// TIA Portal V19 program export: 0 tag tables, 0 data types, 8 data blocks, 13 code blocks (in call order from the OBs), 23 instance data blocks

DATA_BLOCK "AI SCALING DB"   // DB5
{ S7_Optimized_Access := 'TRUE' }
// stored: MemoryReserve 100
   VAR RETAIN
      MIN : Struct
         "SYRUP VESSEL TEMP SENSOR" : Real := -50.0;
         "PREMIXING VESSEL TEMP SENSOR" : Real := -50.0;
         "SUGAR VESSEL TEMP SENSOR" : Real := -50.0;
         "STEAM LINE_1 TEMP SENSOR" : Real := -50.0;
         "STEAM LINE_2 TEMP SENSOR" : Real := -50.0;
         "PRESSURE TRANSMITTER 1" : Real := -1.0;
         "PRESSURE TRANSMITTER 2" : Real := -1.0;
         "VACCIM TRANSMITTER 1" : Real := -750.0;
         "VACCIM TRANSMITTER 2" : Real := -750.0;
         "VACCUM TRANSMITTER 3" : Real := -750.0;
         "SYRUP LOAD CELL" : Real := 0.0;
         "PREMIXING LOAD CELL" : Real := 0.0;
         "SUGAR LOAD CELL" : Real := 0.0;
         "ULTRASONIC LEVEL SENSOR-1" : Real := 0.0;
         "ULTRASONIC LEVEL SENSOR-2" : Real := 0.0;
         "ULTRASONIC LEVEL SENSOR-3" : Real := 0.0;
      END_STRUCT;
      MAX : Struct
         "SYRUP VESSEL TEMP SENSOR" : Real := 250.0;
         "PREMIXING VESSEL TEMP SENSOR" : Real := 250.0;
         "SUGAR VESSEL TEMP SENSOR" : Real := 250.0;
         "STEAM LINE_1 TEMP SENSOR" : Real := 250.0;
         "STEAM LINE_2 TEMP SENSOR" : Real := 250.0;
         "PRESSURE TRANSMITTER 1" : Real := 5.0;
         "PRESSURE TRANSMITTER 2" : Real := 5.0;
         "VACCIM TRANSMITTER 1" : Real := 0.0;
         "VACCIM TRANSMITTER 2" : Real := 0.0;
         "VACCUM TRANSMITTER 3" : Real := 0.0;
         "SYRUP LOAD CELL" : Real := 5000.0;
         "PREMIXING LOAD CELL" : Real := 1500.0;
         "SUGAR LOAD CELL" : Real := 3750.0;
         "ULTRASONIC LEVEL SENSOR-1" : Real := 10000.0;
         "ULTRASONIC LEVEL SENSOR-2" : Real := 10000.0;
         "ULTRASONIC LEVEL SENSOR-3" : Real := 10000.0;
      END_STRUCT;
   END_VAR
   VAR
      PV : Struct
         "SYRUP VESSEL TEMP SENSOR" : Real;
         "PREMIXING VESSEL TEMP SENSOR" : Real;
         "SUGAR VESSEL TEMP SENSOR" : Real;
         "STEAM LINE_1 TEMP SENSOR" : Real;
         "STEAM LINE_2 TEMP SENSOR" : Real;
         "PRESSURE TRANSMITTER 1" : Real;
         "PRESSURE TRANSMITTER 2" : Real;
         "VACCIM TRANSMITTER 1" : Real;
         "VACCIM TRANSMITTER 2" : Real;
         "VACCUM TRANSMITTER 3" : Real;
         "SYRUP LOAD CELL" : Real;
         "PREMIXING LOAD CELL" : Real;
         "SUGAR LOAD CELL" : Real;
         "ULTRASONIC LEVEL SENSOR-1" : Real;
         "ULTRASONIC LEVEL SENSOR-2" : Real;
         "ULTRASONIC LEVEL SENSOR-3" : Real;
      END_STRUCT;
   END_VAR
BEGIN
END_DATA_BLOCK

DATA_BLOCK "AO SCALING DB"   // DB6
{ S7_Optimized_Access := 'TRUE' }
// stored: MemoryReserve 100
   VAR
      SET : Struct
         "SYRUP MFG VESSEL SPEED" : Real;
         "PREMIXING VESSEL SPEED" : Real;
         "SUGAR VESSEL SPEED" : Real;
         SPARE : Real;
      END_STRUCT;
   END_VAR
   VAR RETAIN
      MIN : Struct
         "SYRUP MFG VESSEL SPEED" : Real;
         "PREMIXING VESSEL SPEED" : Real;
         "SUGAR VESSEL SPEED" : Real;
         SPARE : Real;
      END_STRUCT;
      MAX : Struct
         "SYRUP MFG VESSEL SPEED" : Real := 1450.0;
         "PREMIXING VESSEL SPEED" : Real := 1450.0;
         "SUGAR VESSEL SPEED" : Real := 1450.0;
         SPARE : Real;
      END_STRUCT;
   END_VAR
   VAR
      PV : Struct
         "SYRUP MFG VESSEL SPEED" : Real;
         "PREMIXING VESSEL SPEED" : Real;
         "SUGAR VESSEL SPEED" : Real;
         SPARE : Real;
      END_STRUCT;
   END_VAR
BEGIN
END_DATA_BLOCK

DATA_BLOCK "DO MAPING"   // DB2
{ S7_Optimized_Access := 'TRUE' }
// stored: MemoryReserve 100
   VAR
      "SYRUP MFG VESSEL BOTTOM STERROR RUN" : Bool;
      "PREMIXING VESSEL BOTTOM STERROR RUN" : Bool;
      "INLINE 1 HOMOGENIZER MOTOR1 RUN" : Bool;
      "INLINE 2 HOMOGENIZER MOTOR 2 RUN" : Bool;
      "FILTER PRESS MOTOR 1 RUN" : Bool;
      "FILTER PRESS MOTOR 2 RUN" : Bool;
      "VACCUM PUMP MOTOR-W 1 RUN" : Bool;
      "VACCUMP PUMP MOTOR-S2 RUN" : Bool;
      "VACCUMP PUMP MOTOR-W 3 RUN" : Bool;
      "VACCUMP PUMP MOTOR-S 4 RUN" : Bool;
      "SUGAR VESSEL BOTTOM STERROR RUN" : Bool;
      "BASKET FILTER MOTOR RUN" : Bool;
      "PBV-01 INGREDIENT INLET" : Bool;
      "PBV-02 CIP INLET (SPRAY BALL)" : Bool;
      "PBV-03 VENT FILTER ISOLATION" : Bool;
      "PBV-04 PW INLET" : Bool;
      "PBV-07 PREMIX TANK DRAIN VALVE" : Bool;
      "PAV-09 JACKET STEAM INLET" : Bool;
      "PAV-10 JACKET CONDENSATE DRAIN" : Bool;
      "PAV-11 JACKET BYPASS DRAIN VALVE" : Bool;
      "PAV-12 SEAL COOLING INLET" : Bool;
      "PAV-13 WATER COOLING INLET" : Bool;
      "PAV-14 WATER COOLING OUTLET" : Bool;
      "PBV-15 VACUUM INLET" : Bool;
      "PBV-16 VACUUM VENT VALVE" : Bool;
      "PFBV-17 TANK OUTLET VALVE" : Bool;
      "PBV-19 PW INLET" : Bool;
      "PBV-20 CIP INLET (SPRAY BALL)" : Bool;
      "PBV-21 VENT FILTER ISOLATION" : Bool;
      "PBV-22 INGREDIENT INLET (SUGAR INLET)" : Bool;
      "PBV-25 BOTTOM OUTLET TO DRAIN VALVE" : Bool;
      "PAV-27 JACKET STEAM INLET" : Bool;
      "PAV-28 SEAL COOLING INLET" : Bool;
      "PAV-29 JACKET CONDENSATE DRAIN" : Bool;
      "PBV-30 VACUUM INLET VALVE" : Bool;
      "PBV-31 VACUUM VENT VALVE" : Bool;
      "PFBV-32 TANK OUTLET VALVE" : Bool;
      "PBV-36 PW INLET" : Bool;
      "PBV-37 VENT FILTER ISOLATION" : Bool;
      "PBV-38 CIP INLET LINE" : Bool;
      "PBV-41 MFG TANK DRAIN VALVE" : Bool;
      "PAV-50 JACKET STEAM INLET" : Bool;
      "PAV-51 WATER COOLING OUTLET" : Bool;
      "PAV-52 WATER COOLING INLET" : Bool;
      "PAV-53 SEAL COOLING INLET" : Bool;
      "PAV-54 JACKET STEAM OUTLET VALVE" : Bool;
      "PAV-55 JACKET CONDENSATE BYPASS DRAIN" : Bool;
      "PAV-56 INLINE HOMO. SEAL COOLING INLET" : Bool;
      "PBV-57 VACUUM INLET VALVE" : Bool;
      "PFBV-59 TANK OUTLET VALVE" : Bool;
      "PBV-79 BASKET FILTER INLET" : Bool;
      "PBV-80 BOTTOM OUTLET TO BASKET FILTER" : Bool;
      "PBV-81 TANK BOTTOM OUTLET TO CIP OUTLET" : Bool;
      "PBV-82 CIP ISOLATION" : Bool;
      "PBV-83 PREMIX TRANSFER TO MFG VESSEL TRANSFER (TOP DISH)" : Bool;
      "PBV-84 FROM TANK OUTLET TO CIP OUTLET" : Bool;
      "PBV-85 SORBITOL INLET LINE" : Bool;
      "PBV-86 GLUCOSE INLET LINE" : Bool;
      "PBV-87 BASKET FILTER TO PREMIX VESSEL LINE" : Bool;
      "PBV-88 BASKET FILTER TRANSFER LINE" : Bool;
      "PBV-89 BASKET FILTER TO MFG INLET TRANSFER LINE" : Bool;
      "PBV-90 PREMIX TO MFG TRANSFER LINE" : Bool;
      "PBV-91 PREMIX TO MFG TRANSFER LINE" : Bool;
      "PBV-92 PREMIX TO STORAGE – 4 TRANSFER LINE" : Bool;
      "PBV-93 TANK OUTLET TO INLINE HOMOGENIZER LINE" : Bool;
      "PBV-94 INLINE HOMOGENIZER INLET LINE" : Bool;
      "PBV-95 TANK OUTLET TO FILTER PRESS LINE" : Bool;
      "PBV-96 INLINE HOMOGENIZER RECIRCULATION LINE" : Bool;
      "PBV-97 FILTER PRESS OUTLET" : Bool;
      "PBV-98 INLINE HOMOGENIZER TO FILTER PRESS OUTLET LINE" : Bool;
      "PAV-99 INLINE HOMOGENIZER SEAL COOLING" : Bool;
      "PBV-100 FILTER PRESS INLET" : Bool;
      "PBV-101 SUGAR MELTING TO MFG TRANSFER (TOP DISH)" : Bool;
      "PBV-102 PREMIX TO MFG TRANSFER (TOP DISH)" : Bool;
      "PBV-103 CIP INLET (SPRAY BALL)" : Bool;
      "PBV-104 MFG VESSEL TRANSFER LINE" : Bool;
      "PBV-105 INGREDIENT INLET" : Bool;
      "PBV-106 SORBITOL INLET" : Bool;
      "PBV-107 GLUCOSE INLET" : Bool;
      "PBV-108 INLINE HOMOGENIZER TO FILTER PRESS INLET LINE" : Bool;
      "PBV-109 HOMO. RECIRCULATION INLET" : Bool;
      "PBV-110 INLINE HOMOGENIZER TO INLET LINE" : Bool;
      "PBV-111 FILTER PRESS OUTLER VALVE" : Bool;
      "PBV-112 FILTER PRESS TO TRANSFER LINE" : Bool;
      "PAV-113 TANK OUTLET TO CIP DRAIN LINE" : Bool;
      "PBV-114 TANK OUTLET TO INLINE HOMOGENIZER LINE" : Bool;
      "PBV-115 MFG TO STORAGE – 1 TRANSFER LINE" : Bool;
      "PBV-116 MFG TO STORAGE – 2 TRANSFER LINE" : Bool;
      "PBV-117 MFG TO STORAGE – 3 TRANSFER LINE" : Bool;
      "PBV-118 FILTER PRESS INLET" : Bool;
      "PBV-119 SEAL COOLING FOR STORAGE VESSEL - 4" : Bool;
      "PBV-120 SEAL COOLING FOR STORAGE VESSEL - 3" : Bool;
      "PBV-121 SEAL COOLING FOR STORAGE VESSEL - 2" : Bool;
      "PBV-122 SEAL COOLING FOR STORAGE VESSEL - 1" : Bool;
      "PBV-123 VESSEL TOP DISH" : Bool;
      "PBV-124 VESSEL INLET LINE" : Bool;
      "PBV-149" : Bool;
      "PBV-150" : Bool;
      "PBV-151" : Bool;
      "PBV-152" : Bool;
      "PBV-153" : Bool;
      "PBV-155" : Bool;
      "PBV-156" : Bool;
      HOOTER_1 : Bool;
      HOOTR_2 : Bool;
      SPARE_DO1 : Bool;
      SPARE_DO2 : Bool;
      SPARE_DO3 : Bool;
      SPARE_DO4 : Bool;
      SPARE_DO5 : Bool;
      SPARE_DO6 : Bool;
      SPARE_DO7 : Bool;
   END_VAR
BEGIN
END_DATA_BLOCK

DATA_BLOCK "MANUAL TIME BASE DB"   // DB41
{ S7_Optimized_Access := 'TRUE' }
// stored: MemoryReserve 100
   VAR RETAIN
      "MFG VESSEL STIRRER RUN" : Struct
         SV : Int := 555;
         PV : Int := 0;
         "RESET TIME" : Bool := FALSE;
      END_STRUCT;
      "PREMIXING  VESSEL STIRRER RUN" : Struct
         SV : Int := 555;
         PV : Int := 0;
         "RESET TIME" : Bool := FALSE;
      END_STRUCT;
      "SUGAR VESSEL STIRRER RUN" : Struct
         SV : Int := 555;
         PV : Int := 0;
         "RESET TIME" : Bool := FALSE;
      END_STRUCT;
   END_VAR
BEGIN
END_DATA_BLOCK

DATA_BLOCK "TRANSFER DB"   // DB15
{ S7_Optimized_Access := 'TRUE' }
// stored: MemoryReserve 100
   VAR
      "MFG VACCUM PUMP MOTOR-W 1 BIT" : Bool;
      "MFG VACCUMP PUMP MOTOR-S2 BIT" : Bool;
      "PREMIXING VACCUM PUMP MOTOR-W 1 BIT" : Bool;
      "PREMIXING VACCUMP PUMP MOTOR-S2 BIT" : Bool;
      "SUAGR VACCUM PUMP MOTOR-W 3 BIT" : Bool;
      "SUGAR VACCUMP PUMP MOTOR-S4 BIT" : Bool;
      START : Struct
         "SUGAR TO PREMIXING" : Bool;
         "SUGAR TO MFG" : Bool;
         "PREMIXING TO MFG WITH INLINE HOMO" : Bool;
         "PREMIXING TO MFG WITH INLINE FILTER PRES" : Bool;
         "PREMIXING TO STORAGE-4 WITH INLINE HOMO" : Bool;
         "PREMIXING TO STORAGE-4 WITH INLINE FILTER PRES" : Bool;
         "MFG TO STORAGE-1 WITH INLINE HOMO" : Bool;
         "MFG TO STORAGE-1 WITH INLINE FILTER PRES" : Bool;
         "MFG TO STORAGE-2 WITH INLINE HOMO" : Bool;
         "MFG TO STORAGE-2 WITH INLINE FILTER PRES" : Bool;
         "MFG TO STORAGE-3 WITH INLINE HOMO" : Bool;
         "MFG TO STORAGE-3 WITH INLINE FILTER PRES" : Bool;
      END_STRUCT;
      STOP : Struct
         "SUGAR TO PREMIXING" : Bool;
         "SUGAR TO MFG" : Bool;
         "PREMIXING TO MFG WITH INLINE HOMO" : Bool;
         "PREMIXING TO MFG WITH INLINE FILTER PRES" : Bool;
         "PREMIXING TO STORAGE-4 WITH INLINE HOMO" : Bool;
         "PREMIXING TO STORAGE-4 WITH INLINE FILTER PRES" : Bool;
         "MFG TO STORAGE-1 WITH INLINE HOMO" : Bool;
         "MFG TO STORAGE-1 WITH INLINE FILTER PRES" : Bool;
         "MFG TO STORAGE-2 WITH INLINE HOMO" : Bool;
         "MFG TO STORAGE-2 WITH INLINE FILTER PRES" : Bool;
         "MFG TO STORAGE-3 WITH INLINE HOMO" : Bool;
         "MFG TO STORAGE-3 WITH INLINE FILTER PRES" : Bool;
      END_STRUCT;
   END_VAR
   VAR RETAIN
      PAUSE : Struct
         "SUGAR TO PREMIXING" : Bool;
         "SUGAR TO MFG" : Bool;
         "PREMIXING TO MFG WITH INLINE HOMO" : Bool;
         "PREMIXING TO MFG WITH INLINE FILTER PRES" : Bool;
         "PREMIXING TO STORAGE-4 WITH INLINE HOMO" : Bool;
         "PREMIXING TO STORAGE-4 WITH INLINE FILTER PRES" : Bool;
         "MFG TO STORAGE-1 WITH INLINE HOMO" : Bool;
         "MFG TO STORAGE-1 WITH INLINE FILTER PRES" : Bool;
         "MFG TO STORAGE-2 WITH INLINE HOMO" : Bool;
         "MFG TO STORAGE-2 WITH INLINE FILTER PRES" : Bool;
         "MFG TO STORAGE-3 WITH INLINE HOMO" : Bool;
         "MFG TO STORAGE-3 WITH INLINE FILTER PRES" : Bool;
      END_STRUCT;
      BUFF : Struct
         "SUGAR TO PREMIXING" : Int;
         "SUGAR TO MFG" : Int;
         "PREMIXING TO MFG WITH INLINE HOMO" : Int;
         "PREMIXING TO MFG WITH INLINE FILTER PRES" : Int;
         "PREMIXING TO STORAGE-4 WITH INLINE HOMO" : Int;
         "PREMIXING TO STORAGE-4 WITH INLINE FILTER PRES" : Int;
         "MFG TO STORAGE-1 WITH INLINE HOMO" : Int;
         "MFG TO STORAGE-1 WITH INLINE FILTER PRES" : Int;
         "MFG TO STORAGE-2 WITH INLINE HOMO" : Int;
         "MFG TO STORAGE-2 WITH INLINE FILTER PRES" : Int;
         "MFG TO STORAGE-3 WITH INLINE HOMO" : Int;
         "MFG TO STORAGE-3 WITH INLINE FILTER PRES" : Int;
      END_STRUCT;
   END_VAR
   VAR
      BIT : Struct
         "SUGAR TO PREMIXING" : Struct
            "PFBV-32 TANK OUTLET VALVE" : Bool;
            "PBV-80 BOTTOM OUTLET TO BASKET FILTER" : Bool;
            "BASKET FILTER MOTOR RUN" : Bool;
            "PBV-79 BASKET FILTER INLET" : Bool;
            "PBV-149" : Bool;
            "PBV-88 BASKET FILTER TRANSFER LINE" : Bool;
            "PBV-87 BASKET FILTER TO PREMIX VESSEL LINE" : Bool;
         END_STRUCT;
         "SUGAR TO MFG" : Struct
            "PFBV-32 TANK OUTLET VALVE" : Bool;
            "PBV-80 BOTTOM OUTLET TO BASKET FILTER" : Bool;
            "BASKET FILTER MOTOR RUN" : Bool;
            "PBV-79 BASKET FILTER INLET" : Bool;
            "PBV-149" : Bool;
            "PBV-89 BASKET FILTER TO MFG INLET TRANSFER LINE" : Bool;
            "PBV-101 SUGAR MELTING TO MFG TRANSFER (TOP DISH)" : Bool;
         END_STRUCT;
         "PREMIXING TO MFG WITH INLINE HOMO" : Struct
            "PFBV-17 TANK OUTLET VALVE" : Bool;
            "PBV-93 TANK OUTLET TO INLINE HOMOGENIZER LINE" : Bool;
            "PBV-94 INLINE HOMOGENIZER INLET LINE" : Bool;
            "PAV-99 INLINE HOMOGENIZER SEAL COOLING" : Bool;
            "INLINE 2 HOMOGENIZER MOTOR 2 RUN" : Bool;
            "PBV-96 INLINE HOMOGENIZER RECIRCULATION LINE" : Bool;
            "PBV-91 PREMIX TO MFG TRANSFER LINE" : Bool;
            "PBV-102 PREMIX TO MFG TRANSFER (TOP DISH)" : Bool;
         END_STRUCT;
         "PREMIXING TO MFG WITH INLINE FILTER PRES" : Struct
            "PFBV-17 TANK OUTLET VALVE" : Bool;
            "PBV-93 TANK OUTLET TO INLINE HOMOGENIZER LINE" : Bool;
            "PBV-95 TANK OUTLET TO FILTER PRESS LINE" : Bool;
            "FILTER PRESS MOTOR 2 RUN" : Bool;
            "PBV-100 FILTER PRESS INLET" : Bool;
            "PBV-97 FILTER PRESS OUTLET" : Bool;
            "PBV-98 INLINE HOMOGENIZER TO FILTER PRESS OUTLET LINE" : Bool;
            "PBV-91 PREMIX TO MFG TRANSFER LINE" : Bool;
            "PBV-102 PREMIX TO MFG TRANSFER (TOP DISH)" : Bool;
         END_STRUCT;
         "PREMIXING TO STORAGE-4 WITH INLINE HOMO" : Struct
            "PFBV-17 TANK OUTLET VALVE" : Bool;
            "PBV-93 TANK OUTLET TO INLINE HOMOGENIZER LINE" : Bool;
            "PBV-94 INLINE HOMOGENIZER INLET LINE" : Bool;
            "PAV-99 INLINE HOMOGENIZER SEAL COOLING" : Bool;
            "INLINE 2 HOMOGENIZER MOTOR 2 RUN" : Bool;
            "PBV-96 INLINE HOMOGENIZER RECIRCULATION LINE" : Bool;
            "PBV-92 PREMIX TO STORAGE – 4 TRANSFER LINE" : Bool;
         END_STRUCT;
         "PREMIXING TO STORAGE-4 WITH INLINE FILTER PRES" : Struct
            "PFBV-17 TANK OUTLET VALVE" : Bool;
            "PBV-93 TANK OUTLET TO INLINE HOMOGENIZER LINE" : Bool;
            "PBV-95 TANK OUTLET TO FILTER PRESS LINE" : Bool;
            "FILTER PRESS MOTOR 2 RUN" : Bool;
            "PBV-100 FILTER PRESS INLET" : Bool;
            "PBV-97 FILTER PRESS OUTLET" : Bool;
            "PBV-98 INLINE HOMOGENIZER TO FILTER PRESS OUTLET LINE" : Bool;
            "PBV-92 PREMIX TO STORAGE – 4 TRANSFER LINE" : Bool;
         END_STRUCT;
         "MFG TO STORAGE-1 WITH INLINE HOMO" : Struct
            "PFBV-59 TANK OUTLET VALVE" : Bool;
            "PBV-114 TANK OUTLET TO INLINE HOMOGENIZER LINE" : Bool;
            "PBV-110 INLINE HOMOGENIZER TO INLET LINE" : Bool;
            "PAV-56 INLINE HOMO. SEAL COOLING INLET" : Bool;
            "INLINE 1 HOMOGENIZER MOTOR1 RUN" : Bool;
            "PBV-109 HOMO. RECIRCULATION INLET" : Bool;
            "PBV-115 MFG TO STORAGE – 1 TRANSFER LINE" : Bool;
         END_STRUCT;
         "MFG TO STORAGE-1 WITH INLINE FILTER PRES" : Struct
            "PFBV-59 TANK OUTLET VALVE" : Bool;
            "PBV-114 TANK OUTLET TO INLINE HOMOGENIZER LINE" : Bool;
            "PBV-108 INLINE HOMOGENIZER TO FILTER PRESS INLET LINE" : Bool;
            "FILTER PRESS MOTOR 1 RUN" : Bool;
            "PBV-118 FILTER PRESS INLET" : Bool;
            "PBV-111 FILTER PRESS OUTLER VALVE" : Bool;
            "PBV-112 FILTER PRESS TO TRANSFER LINE" : Bool;
            "PBV-115 MFG TO STORAGE – 1 TRANSFER LINE" : Bool;
         END_STRUCT;
         "MFG TO STORAGE-2 WITH INLINE HOMO" : Struct
            "PFBV-59 TANK OUTLET VALVE" : Bool;
            "PBV-114 TANK OUTLET TO INLINE HOMOGENIZER LINE" : Bool;
            "PBV-110 INLINE HOMOGENIZER TO INLET LINE" : Bool;
            "PAV-56 INLINE HOMO. SEAL COOLING INLET" : Bool;
            "INLINE 1 HOMOGENIZER MOTOR1 RUN" : Bool;
            "PBV-109 HOMO. RECIRCULATION INLET" : Bool;
            "PBV-116 MFG TO STORAGE – 2 TRANSFER LINE" : Bool;
         END_STRUCT;
         "MFG TO STORAGE-2 WITH INLINE FILTER PRES" : Struct
            "PFBV-59 TANK OUTLET VALVE" : Bool;
            "PBV-114 TANK OUTLET TO INLINE HOMOGENIZER LINE" : Bool;
            "PBV-108 INLINE HOMOGENIZER TO FILTER PRESS INLET LINE" : Bool;
            "FILTER PRESS MOTOR 1 RUN" : Bool;
            "PBV-118 FILTER PRESS INLET" : Bool;
            "PBV-111 FILTER PRESS OUTLER VALVE" : Bool;
            "PBV-112 FILTER PRESS TO TRANSFER LINE" : Bool;
            "PBV-116 MFG TO STORAGE – 2 TRANSFER LINE" : Bool;
         END_STRUCT;
         "MFG TO STORAGE-3 WITH INLINE HOMO" : Struct
            "PFBV-59 TANK OUTLET VALVE" : Bool;
            "PBV-114 TANK OUTLET TO INLINE HOMOGENIZER LINE" : Bool;
            "PBV-110 INLINE HOMOGENIZER TO INLET LINE" : Bool;
            "PAV-56 INLINE HOMO. SEAL COOLING INLET" : Bool;
            "INLINE 1 HOMOGENIZER MOTOR1 RUN" : Bool;
            "PBV-109 HOMO. RECIRCULATION INLET" : Bool;
            "PBV-117 MFG TO STORAGE – 3 TRANSFER LINE" : Bool;
         END_STRUCT;
         "MFG TO STORAGE-3 WITH INLINE FILTER PRES" : Struct
            "PFBV-59 TANK OUTLET VALVE" : Bool;
            "PBV-114 TANK OUTLET TO INLINE HOMOGENIZER LINE" : Bool;
            "PBV-108 INLINE HOMOGENIZER TO FILTER PRESS INLET LINE" : Bool;
            "FILTER PRESS MOTOR 1 RUN" : Bool;
            "PBV-118 FILTER PRESS INLET" : Bool;
            "PBV-111 FILTER PRESS OUTLER VALVE" : Bool;
            "PBV-112 FILTER PRESS TO TRANSFER LINE" : Bool;
            "PBV-117 MFG TO STORAGE – 3 TRANSFER LINE" : Bool;
         END_STRUCT;
      END_STRUCT;
      OUTPUT : Struct
         "SYRUP MFG VESSEL BOTTOM STERROR RUN" : Bool;
         "PREMIXING VESSEL BOTTOM STERROR RUN" : Bool;
         "INLINE 1 HOMOGENIZER MOTOR1 RUN" : Bool;
         "INLINE 2 HOMOGENIZER MOTOR 2 RUN" : Bool;
         "FILTER PRESS MOTOR 1 RUN" : Bool;
         "FILTER PRESS MOTOR 2 RUN" : Bool;
         "VACCUM PUMP MOTOR-W 1 RUN" : Bool;
         "VACCUMP PUMP MOTOR-S2 RUN" : Bool;
         "VACCUMP PUMP MOTOR-W 3 RUN" : Bool;
         "VACCUMP PUMP MOTOR-S 4 RUN" : Bool;
         "SUGAR VESSEL BOTTOM STERROR RUN" : Bool;
         "BASKET FILTER MOTOR RUN" : Bool;
         "PBV-01 INGREDIENT INLET" : Bool;
         "PBV-02 CIP INLET (SPRAY BALL)" : Bool;
         "PBV-03 VENT FILTER ISOLATION" : Bool;
         "PBV-04 PW INLET" : Bool;
         "PBV-07 PREMIX TANK DRAIN VALVE" : Bool;
         "PAV-09 JACKET STEAM INLET" : Bool;
         "PAV-10 JACKET CONDENSATE DRAIN" : Bool;
         "PAV-11 JACKET BYPASS DRAIN VALVE" : Bool;
         "PAV-12 SEAL COOLING INLET" : Bool;
         "PAV-13 WATER COOLING INLET" : Bool;
         "PAV-14 WATER COOLING OUTLET" : Bool;
         "PBV-15 VACUUM INLET" : Bool;
         "PBV-16 VACUUM VENT VALVE" : Bool;
         "PFBV-17 TANK OUTLET VALVE" : Bool;
         "PBV-19 PW INLET" : Bool;
         "PBV-20 CIP INLET (SPRAY BALL)" : Bool;
         "PBV-21 VENT FILTER ISOLATION" : Bool;
         "PBV-22 INGREDIENT INLET (SUGAR INLET)" : Bool;
         "PBV-25 BOTTOM OUTLET TO DRAIN VALVE" : Bool;
         "PAV-27 JACKET STEAM INLET" : Bool;
         "PAV-28 SEAL COOLING INLET" : Bool;
         "PAV-29 JACKET CONDENSATE DRAIN" : Bool;
         "PBV-30 VACUUM INLET VALVE" : Bool;
         "PBV-31 VACUUM VENT VALVE" : Bool;
         "PFBV-32 TANK OUTLET VALVE" : Bool;
         "PBV-36 PW INLET" : Bool;
         "PBV-37 VENT FILTER ISOLATION" : Bool;
         "PBV-38 CIP INLET LINE" : Bool;
         "PBV-41 MFG TANK DRAIN VALVE" : Bool;
         "PAV-50 JACKET STEAM INLET" : Bool;
         "PAV-51 WATER COOLING OUTLET" : Bool;
         "PAV-52 WATER COOLING INLET" : Bool;
         "PAV-53 SEAL COOLING INLET" : Bool;
         "PAV-54 JACKET STEAM OUTLET VALVE" : Bool;
         "PAV-55 JACKET CONDENSATE BYPASS DRAIN" : Bool;
         "PAV-56 INLINE HOMO. SEAL COOLING INLET" : Bool;
         "PBV-57 VACUUM INLET VALVE" : Bool;
         "PFBV-59 TANK OUTLET VALVE" : Bool;
         "PBV-79 BASKET FILTER INLET" : Bool;
         "PBV-80 BOTTOM OUTLET TO BASKET FILTER" : Bool;
         "PBV-81 TANK BOTTOM OUTLET TO CIP OUTLET" : Bool;
         "PBV-82 CIP ISOLATION" : Bool;
         "PBV-83 PREMIX TRANSFER TO MFG VESSEL TRANSFER (TOP DISH)" : Bool;
         "PBV-84 FROM TANK OUTLET TO CIP OUTLET" : Bool;
         "PBV-85 SORBITOL INLET LINE" : Bool;
         "PBV-86 GLUCOSE INLET LINE" : Bool;
         "PBV-87 BASKET FILTER TO PREMIX VESSEL LINE" : Bool;
         "PBV-88 BASKET FILTER TRANSFER LINE" : Bool;
         "PBV-89 BASKET FILTER TO MFG INLET TRANSFER LINE" : Bool;
         "PBV-90 PREMIX TO MFG TRANSFER LINE" : Bool;
         "PBV-91 PREMIX TO MFG TRANSFER LINE" : Bool;
         "PBV-92 PREMIX TO STORAGE – 4 TRANSFER LINE" : Bool;
         "PBV-93 TANK OUTLET TO INLINE HOMOGENIZER LINE" : Bool;
         "PBV-94 INLINE HOMOGENIZER INLET LINE" : Bool;
         "PBV-95 TANK OUTLET TO FILTER PRESS LINE" : Bool;
         "PBV-96 INLINE HOMOGENIZER RECIRCULATION LINE" : Bool;
         "PBV-97 FILTER PRESS OUTLET" : Bool;
         "PBV-98 INLINE HOMOGENIZER TO FILTER PRESS OUTLET LINE" : Bool;
         "PAV-99 INLINE HOMOGENIZER SEAL COOLING" : Bool;
         "PBV-100 FILTER PRESS INLET" : Bool;
         "PBV-101 SUGAR MELTING TO MFG TRANSFER (TOP DISH)" : Bool;
         "PBV-102 PREMIX TO MFG TRANSFER (TOP DISH)" : Bool;
         "PBV-103 CIP INLET (SPRAY BALL)" : Bool;
         "PBV-104 MFG VESSEL TRANSFER LINE" : Bool;
         "PBV-105 INGREDIENT INLET" : Bool;
         "PBV-106 SORBITOL INLET" : Bool;
         "PBV-107 GLUCOSE INLET" : Bool;
         "PBV-108 INLINE HOMOGENIZER TO FILTER PRESS INLET LINE" : Bool;
         "PBV-109 HOMO. RECIRCULATION INLET" : Bool;
         "PBV-110 INLINE HOMOGENIZER TO INLET LINE" : Bool;
         "PBV-111 FILTER PRESS OUTLER VALVE" : Bool;
         "PBV-112 FILTER PRESS TO TRANSFER LINE" : Bool;
         "PAV-113 TANK OUTLET TO CIP DRAIN LINE" : Bool;
         "PBV-114 TANK OUTLET TO INLINE HOMOGENIZER LINE" : Bool;
         "PBV-115 MFG TO STORAGE – 1 TRANSFER LINE" : Bool;
         "PBV-116 MFG TO STORAGE – 2 TRANSFER LINE" : Bool;
         "PBV-117 MFG TO STORAGE – 3 TRANSFER LINE" : Bool;
         "PBV-118 FILTER PRESS INLET" : Bool;
         "PBV-119 SEAL COOLING FOR STORAGE VESSEL - 4" : Bool;
         "PBV-120 SEAL COOLING FOR STORAGE VESSEL - 3" : Bool;
         "PBV-121 SEAL COOLING FOR STORAGE VESSEL - 2" : Bool;
         "PBV-122 SEAL COOLING FOR STORAGE VESSEL - 1" : Bool;
         "PBV-123 VESSEL TOP DISH" : Bool;
         "PBV-124 VESSEL INLET LINE" : Bool;
         "PBV-149" : Bool;
         "PBV-150" : Bool;
         "PBV-151" : Bool;
         "PBV-152" : Bool;
         "PBV-153" : Bool;
         "PBV-155" : Bool;
         "PBV-156" : Bool;
         HOOTER_1 : Bool;
         HOOTR_2 : Bool;
      END_STRUCT;
   END_VAR
BEGIN
END_DATA_BLOCK

DATA_BLOCK "AUTO ALARM DB"   // DB70
{ S7_Optimized_Access := 'TRUE' }
// stored: MemoryReserve 100
   VAR
      "MFG PROCESS" : Struct
         "PURIFIED WATER PROCESS SELECT" : Bool;
         "PURIFIED WATER PROCESS OF INITIAL DRAIN SELECT" : Bool;
         "PURIFIED WATER PROCESS OF LOAD CELL" : Bool;
         "PURIFIED WATER HEATING OR COOLING SELECT" : Bool;
         "PURIFIED WATER PROCESS OF JACKET DRAIN SELECT" : Bool;
         "PURIFIED WATER PROCESS OVER" : Bool;
         "MATERIAL ADDITION PROCESS SELECT" : Bool;
         "MATERIAL ADDITION MATERIAL ADDED TEXT" : Bool;
         "MATERIAL ADDITION DO YOU WANT TO ADD SORBITOL SELECT" : Bool;
         "MATERIAL ADDITION OF SORBITOL OVER" : Bool;
         "MATERIAL ADDITION DO YOU WANT TO ADD GLUCOSE SELECT" : Bool;
         "MATERIAL ADDITION OF GLUCOSE OVER" : Bool;
         "MATERIAL ADDITION PROCESS OVER" : Bool;
         "RECIRCULATION PROCESS SELECT" : Bool;
         "RECIRCULATION PROCESS RUNING" : Bool;
         "RECIRCULATION OVER" : Bool;
         "MFG PROCESS OVER" : Bool;
      END_STRUCT;
      "MFG PROCESS ALARM" : Struct
         "MFG PROCESS START" : Bool;
         "PURIFIED WATER PROCESS START" : Bool;
         "PURIFIED WATER PROCESS OF INITIAL DRAIN START" : Bool;
         "PURIFIED WATER PROCESS OF INITIAL DRAIN STOP" : Bool;
         "PURIFIED WATER PROCESS OF LOAD CELL START" : Bool;
         "PURIFIED WATER PROCESS OF LOAD CELL STOP" : Bool;
         "PURIFIED WATER OF HEATING START" : Bool;
         "PURIFIED WATER OF HEATING STOP" : Bool;
         "PURIFIED WATER OF COOLING START" : Bool;
         "PURIFIED WATER OF COOLING STOP" : Bool;
         "PURIFIED WATER PROCESS OF JACKET DRAIN START" : Bool;
         "PURIFIED WATER PROCESS OF JACKET DRAIN STOP" : Bool;
         "PURIFIED WATER PROCESS OVER" : Bool;
         "MATERIAL ADDITION PROCESS START" : Bool;
         "MATERIAL ADDITION MATERIAL ADDED TEXT" : Bool;
         "MATERIAL ADDITION OF SORBITOL START" : Bool;
         "MATERIAL ADDITION OF SORBITOL OVER" : Bool;
         "MATERIAL ADDITION OF GLUCOSE START" : Bool;
         "MATERIAL ADDITION OF GLUCOSE OVER" : Bool;
         "MATERIAL ADDITION PROCESS OVER" : Bool;
         "RECIRCULATION PROCESS START" : Bool;
         "RECIRCULATION PROCESS OVER" : Bool;
         "MFG PROCESS OVER" : Bool;
      END_STRUCT;
      "MFG TRANSFER START" : Struct
         "MFG TO STORAGE-1 WITH INLINE HOMO" : Bool;
         "MFG TO STORAGE-1 WITH INLINE FILTER PRES" : Bool;
         "MFG TO STORAGE-2 WITH INLINE HOMO" : Bool;
         "MFG TO STORAGE-2 WITH INLINE FILTER PRES" : Bool;
         "MFG TO STORAGE-3 WITH INLINE HOMO" : Bool;
         "MFG TO STORAGE-3 WITH INLINE FILTER PRES" : Bool;
      END_STRUCT;
      "MFG TRANSFER OVER" : Struct
         "TRANSFER START_MFG TO STORAGE ALL IN ONE FOR OVER (POPUP)" : Bool;
         "MFG TO STORAGE-1 WITH INLINE HOMO" : Bool;
         "MFG TO STORAGE-1 WITH INLINE FILTER PRES" : Bool;
         "MFG TO STORAGE-2 WITH INLINE HOMO" : Bool;
         "MFG TO STORAGE-2 WITH INLINE FILTER PRES" : Bool;
         "MFG TO STORAGE-3 WITH INLINE HOMO" : Bool;
         "MFG TO STORAGE-3 WITH INLINE FILTER PRES" : Bool;
      END_STRUCT;
      "MFG MATERIAL SUCTION" : Struct
         "MATERIAL SUCTION START" : Bool;
         "MATERIAL SUCTION OVER" : Bool;
      END_STRUCT;
      "PREMIXING PROCESS" : Struct
         "PURIFIED WATER PROCESS SELECT" : Bool;
         "PURIFIED WATER PROCESS OF INITIAL DRAIN SELECT" : Bool;
         "PURIFIED WATER PROCESS OF LOAD CELL" : Bool;
         "PURIFIED WATER HEATING OR COOLING SELECT" : Bool;
         "PURIFIED WATER PROCESS OF JACKET DRAIN SELECT" : Bool;
         "PURIFIED WATER PROCESS OVER" : Bool;
         "MATERIAL ADDITION PROCESS SELECT" : Bool;
         "MATERIAL ADDITION MATERIAL ADDED TEXT" : Bool;
         "MATERIAL ADDITION DO YOU WANT TO ADD SORBITOL SELECT" : Bool;
         "MATERIAL ADDITION OF SORBITOL OVER" : Bool;
         "MATERIAL ADDITION DO YOU WANT TO ADD GLUCOSE SELECT" : Bool;
         "MATERIAL ADDITION OF GLUCOSE OVER" : Bool;
         "MATERIAL ADDITION PROCESS OVER" : Bool;
         "RECIRCULATION PROCESS SELECT" : Bool;
         "RECIRCULATION PROCESS RUNING" : Bool;
         "RECIRCULATION OVER" : Bool;
         "PREMIXING PROCESS OVER" : Bool;
      END_STRUCT;
      "PREMIXING PROCESS ALARM" : Struct
         "PREMIXING PROCESS START" : Bool;
         "PURIFIED WATER PROCESS START" : Bool;
         "PURIFIED WATER PROCESS OF INITIAL DRAIN START" : Bool;
         "PURIFIED WATER PROCESS OF INITIAL DRAIN STOP" : Bool;
         "PURIFIED WATER PROCESS OF LOAD CELL START" : Bool;
         "PURIFIED WATER PROCESS OF LOAD CELL STOP" : Bool;
         "PURIFIED WATER OF HEATING START" : Bool;
         "PURIFIED WATER OF HEATING STOP" : Bool;
         "PURIFIED WATER OF COOLING START" : Bool;
         "PURIFIED WATER OF COOLING STOP" : Bool;
         "PURIFIED WATER PROCESS OF JACKET DRAIN START" : Bool;
         "PURIFIED WATER PROCESS OF JACKET DRAIN STOP" : Bool;
         "PURIFIED WATER PROCESS OVER" : Bool;
         "MATERIAL ADDITION PROCESS START" : Bool;
         "MATERIAL ADDITION OF INITIAL DRAIN START" : Bool;
         "MATERIAL ADDITION OF INITIAL DRAIN STOP" : Bool;
         "MATERIAL ADDITION MATERIAL ADDED TEXT" : Bool;
         "MATERIAL ADDITION OF SORBITOL START" : Bool;
         "MATERIAL ADDITION OF SORBITOL OVER" : Bool;
         "MATERIAL ADDITION OF GLUCOSE START" : Bool;
         "MATERIAL ADDITION OF GLUCOSE OVER" : Bool;
         "MATERIAL ADDITION PROCESS OF JACKET DRAIN SELECT" : Bool;
         "MATERIAL ADDITION PROCESS OF JACKET DRAIN STOP" : Bool;
         "MATERIAL ADDITION PROCESS OVER" : Bool;
         "RECIRCULATION PROCESS START" : Bool;
         "RECIRCULATION PROCESS OF INITIAL DRAIN START" : Bool;
         "RECIRCULATION PROCESS OF INITIAL DRAIN STOP" : Bool;
         "RECIRCULATION START" : Bool;
         "RECIRCULATION STOP" : Bool;
         "RECIRCULATION PROCESS OF JACKET DRAIN SELECT" : Bool;
         "RECIRCULATION PROCESS OF JACKET DRAIN STOP" : Bool;
         "RECIRCULATION PROCESS OVER" : Bool;
         "PREMIXING PROCESS OVER" : Bool;
      END_STRUCT;
      "PREMIXING TRANSFER START" : Struct
         "PREMIXING TO MFG WITH INLINE HOMO" : Bool;
         "PREMIXING TO MFG WITH INLINE FILTER PRES" : Bool;
         "PREMIXING TO STORAGE-4 WITH INLINE HOMO" : Bool;
         "PREMIXING TO STORAGE-4 WITH INLINE FILTER PRES" : Bool;
      END_STRUCT;
      "PREMIXING TRANSFER OVER" : Struct
         "PREMIXING TO MFG & STORAGE ALL IN ONE FOR OVER (POPUP)" : Bool;
         "PREMIXING TO MFG WITH INLINE HOMO" : Bool;
         "PREMIXING TO MFG WITH INLINE FILTER PRES" : Bool;
         "PREMIXING TO STORAGE-4 WITH INLINE HOMO" : Bool;
         "PREMIXING TO STORAGE-4 WITH INLINE FILTER PRES" : Bool;
      END_STRUCT;
      "PREMIXING MATERIAL SUCTION" : Struct
         "MATERIAL SUCTION START" : Bool;
         "MATERIAL SUCTION OVER" : Bool;
      END_STRUCT;
      "SUGAR PROCESS" : Struct
         "PURIFIED WATER PROCESS SELECT" : Bool;
         "PURIFIED WATER PROCESS OF INITIAL DRAIN SELECT" : Bool;
         "PURIFIED WATER PROCESS OF LOAD CELL" : Bool;
         "PURIFIED WATER HEATING OR COOLING SELECT" : Bool;
         "PURIFIED WATER PROCESS OF JACKET DRAIN SELECT" : Bool;
         "PURIFIED WATER PROCESS OVER" : Bool;
         "MFG PROCESS OVER" : Bool;
      END_STRUCT;
      "SUGAR PROCESS ALARM" : Struct
         "SUGAR PROCESS START" : Bool;
         "PURIFIED WATER PROCESS START" : Bool;
         "PURIFIED WATER PROCESS OF INITIAL DRAIN START" : Bool;
         "PURIFIED WATER PROCESS OF INITIAL DRAIN STOP" : Bool;
         "PURIFIED WATER PROCESS OF LOAD CELL START" : Bool;
         "PURIFIED WATER PROCESS OF LOAD CELL STOP" : Bool;
         "PURIFIED WATER OF HEATING START" : Bool;
         "PURIFIED WATER OF HEATING STOP" : Bool;
         "PURIFIED WATER OF COOLING START" : Bool;
         "PURIFIED WATER OF COOLING STOP" : Bool;
         "PURIFIED WATER PROCESS OF JACKET DRAIN START" : Bool;
         "PURIFIED WATER PROCESS OF JACKET DRAIN STOP" : Bool;
         "PURIFIED WATER PROCESS OVER" : Bool;
      END_STRUCT;
      "SUGAR TRANSFER START" : Struct
         "SUGAR TRANSFER SELECT POPUP" : Bool;
         "TRANSFER PREMIXING AND MFG POPUP" : Bool;
         "SUGAR TO PREMIXING" : Bool;
         "SUGAR TO MFG" : Bool;
      END_STRUCT;
      "SUGAR TRANSFER OVER" : Struct
         "SUGAR TRANSFER OVER POPUP" : Bool;
         "SUGAR TO PREMIXING" : Bool;
         "SUGAR TO MFG" : Bool;
      END_STRUCT;
      "SUGAR MATERIAL SUCTION" : Struct
         "MATERIAL SUCTION START" : Bool;
         "MATERIAL SUCTION OVER" : Bool;
      END_STRUCT;
   END_VAR
BEGIN
END_DATA_BLOCK

DATA_BLOCK "MANUAL INTERLOCK DB"   // DB7
{ S7_Optimized_Access := 'TRUE' }
// stored: MemoryReserve 100
   VAR
      "MAIN ERROR" : Bool;
      "SYRUP MFG UNHEALTHY" : Int;
      "PREMIXING UNHEALTHY" : Int;
      "SUGAR UNHEALTHY" : Int;
      "MFG TRANSFER PROCESS INTERLOCK" : Int;
      "PREMIXING TRANSFER PROCESS INTERLOCK" : Int;
      "SUGAR TRANSFER PROCESS INTERLOCK" : Int;
   END_VAR
BEGIN
END_DATA_BLOCK

DATA_BLOCK "MFG PROCESS_DB"   // DB45
{ S7_Optimized_Access := 'TRUE' }
// stored: MemoryReserve 100
   VAR
      START : Bool;
   END_VAR
   VAR RETAIN
      PAUSE : Bool;
   END_VAR
   VAR
      STOP : Bool;
   END_VAR
   VAR RETAIN
      "AUTO BUFF" : Int;
   END_VAR
   VAR
      "MFG PROCESS OVER" : Bool;
      BIT : Struct
         "PURIFIED WATER" : Struct
            "PURIFIED WATER SELECT" : Bool;
            "PURIFIED WATER SKIP" : Bool;
            "PURIFIED WATER PROCESS OF INITIAL DRAIN SELECT" : Bool;
            "PURIFIED WATER PROCESS OF INITIAL DRAIN SKIP" : Bool;
            "PURIFIED WATER LOAD CELL" : Bool;
            "SELECT HEATING" : Bool;
            "SELECT COOLING" : Bool;
            "PURIFIED WATER OVER" : Bool;
            "PURIFIED WATER PROCESS OF JACKET DRAIN SELECT" : Bool;
            "PURIFIED WATER PROCESS OF JACKET DRAIN SKIP" : Bool;
         END_STRUCT;
         "MATERIAL ADDITION" : Struct
            "MATERIAL SELECT" : Bool;
            "MATERIAL SKIP" : Bool;
            "MATERIAL ADDED" : Bool;
            "SORBITOL SELECT" : Bool;
            "SORBITOL SKIP" : Bool;
            "SORBITOL OVER" : Bool;
            "GLUCOSE SELECT" : Bool;
            "GLUCOSE SKIP" : Bool;
            "GLUCOSE OVER" : Bool;
            "MATERIAL OVER" : Bool;
         END_STRUCT;
         RECIRCULATION : Struct
            "RECIRCULATION SEL" : Bool;
            "RECIRCULATION SKIP" : Bool;
            "RECIRCULATION START" : Bool;
            "RECIRCULATION OVER" : Bool;
         END_STRUCT;
      END_STRUCT;
   END_VAR
   VAR RETAIN
      "MATERIAL SUCTION" : Struct
         "MATERIAL SUCTION START" : Bool;
         "MATERIAL SUCTION STOP" : Bool;
         "MATERIAL SUCTION OVER" : Bool;
         "MATERIAL SUCTION BUFF" : Int;
      END_STRUCT;
      "SET PARAMETER" : Struct
         "PURIFIED WATER INITIAL DRAIN TIME" : Int;
         "PURIFIED LOAD" : Real;
         "PURIFIED HEATING" : Real;
         "PURIFIED COOLING" : Real;
         "PURIFIED STIRRER MOTOR RPM" : Real;
         "PURIFIED STIRRER_TIME" : Int;
         "PURIFIED WATER JACKET DRAIN TIME" : Int;
         "MATERIAL_SORBITOL LOAD CELL" : Real;
         "MATERIAL_SORBITOL STIRRER TIME" : Int;
         "MATERIAL SORBITOL STIRRER MOTOR RPM" : Real;
         "MATERIAL_SORBITOL TEMP_MAX" : Real;
         "MATERIAL_SORBITOL TEMP_MIN" : Real;
         "MATERIAL_GLUCOSE LOAD CELL" : Real;
         "MATERIAL_GLUCOSE STIRRER TIME" : Int;
         "MATERIAL GLUCOSE STIRRER MOTOR RPM" : Real;
         "MATERIAL_GLUCOSE TEMP_MAX" : Real;
         "MATERIAL_GLUCOSE TEMP_MIN" : Real;
         "RECIRCULATION TOTAL TIME" : Int;
         "RECIRCULATION STIRRER RPM" : Real;
         "RECIRCULATION HOMOGENIZER DELAY" : Int;
         "MATERIAL SUCTION VACUUM HIGH" : Real;
         "MATERIAL SUCTION VACUUM LOW" : Real;
         "MATERIAL SUCTION STIRRER RPM" : Real;
         "MATERIAL SUCTION LOAD CELL" : Real;
      END_STRUCT;
      "PV PARAMETER" : Struct
         "PURIFIED WATER INITIAL DRAIN TIME" : Int;
         "PURIFIED STIRRER_TIME" : Int;
         "PURIFIED WATER JACKET DRAIN TIME" : Int;
         "MATERIAL_SORBITOL STIRRER TIME" : Int;
         "MATERIAL_GLUCOSE STIRRER TIME" : Int;
         "RECIRCULATION TOTAL TIME" : Int;
         "RECIRCULATION HOMOGENIZER DELAY" : Int;
         "PURIFIED LOAD" : Real;
         "MATERIAL_SORBITOL LOAD CELL" : Real;
         "MATERIAL_GLUCOSE LOAD CELL" : Real;
         "MATERIAL SUCTION LOAD CELL" : Real;
      END_STRUCT;
   END_VAR
BEGIN
END_DATA_BLOCK

ORGANIZATION_BLOCK "Main"   // OB1, LAD, ProgramCycle
TITLE = "Main Program Sweep (Cycle)"
{ S7_Optimized_Access := 'TRUE' }
// stored: SetENOAutomatically false
   VAR_INPUT
      Initial_Call : Bool;   // Initial call of this OB
      Remanence : Bool;   // =True, if remanent data are available
   END_VAR
   VAR_TEMP   // added for the SCL form of the ladder/FBD networks
      _w1 : Bool;
      _w2 : Bool;
      _w3 : Bool;
      _w4 : Bool;
      _w5 : Bool;
      _w6 : Bool;
      _w7 : Bool;
      _w8 : Bool;
      _w9 : Bool;
      _w10 : Bool;
   END_VAR
BEGIN

REGION Network 1: #SHIV
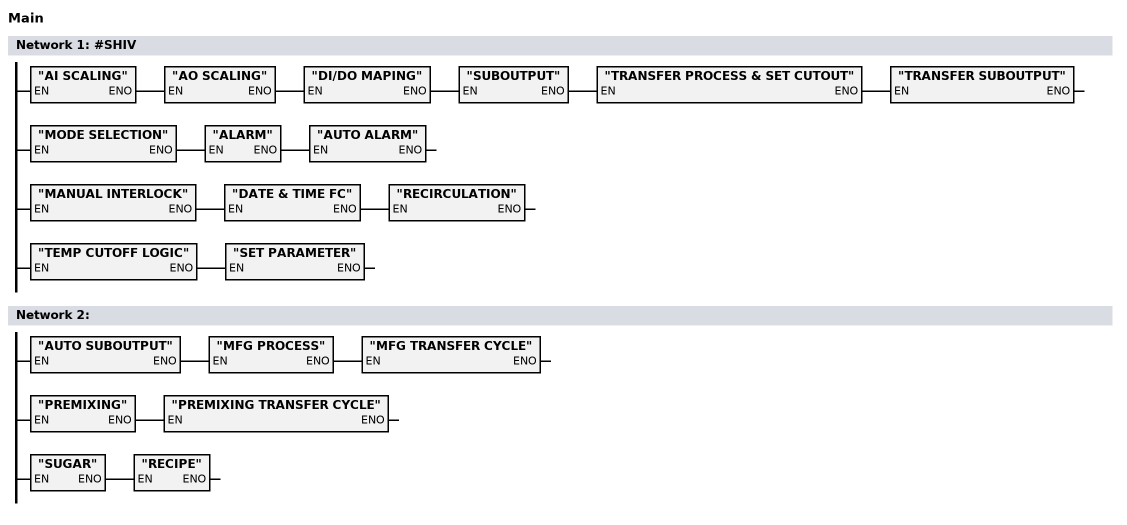
   RUNG wire#powerrail
      "AI SCALING"()
      "AO SCALING"()
      "DI/DO MAPING"()
      "SUBOUTPUT"()
      "TRANSFER PROCESS & SET CUTOUT"()
      "TRANSFER SUBOUTPUT"()
   END_RUNG
   RUNG wire#powerrail
      "MODE SELECTION"()
      "ALARM"()
      "AUTO ALARM"()
   END_RUNG
   RUNG wire#powerrail
      "MANUAL INTERLOCK"()
      "DATE & TIME FC"()
      "RECIRCULATION"()
   END_RUNG
   RUNG wire#powerrail
      "TEMP CUTOFF LOGIC"()
      "SET PARAMETER"()
   END_RUNG
   // the same network as SCL:
   "AI SCALING"(ENO => #_w1);
   "AO SCALING"(EN := #_w1, ENO => #_w2);
   "DI/DO MAPING"(EN := #_w2, ENO => #_w3);
   "SUBOUTPUT"(EN := #_w3, ENO => #_w4);
   "TRANSFER PROCESS & SET CUTOUT"(EN := #_w4, ENO => #_w5);
   IF #_w5 THEN "TRANSFER SUBOUTPUT"(); END_IF;
   "MODE SELECTION"(ENO => #_w6);
   "ALARM"(EN := #_w6, ENO => #_w7);
   IF #_w7 THEN "AUTO ALARM"(); END_IF;
   "MANUAL INTERLOCK"(ENO => #_w8);
   "DATE & TIME FC"(EN := #_w8, ENO => #_w9);
   IF #_w9 THEN "RECIRCULATION"(); END_IF;
   "TEMP CUTOFF LOGIC"(ENO => #_w10);
   IF #_w10 THEN "SET PARAMETER"(); END_IF;
END_REGION

REGION Network 2
   RUNG wire#powerrail
      "AUTO SUBOUTPUT"()
      "MFG PROCESS"()
      "MFG TRANSFER CYCLE"()
   END_RUNG
   RUNG wire#powerrail
      "PREMIXING"()
      "PREMIXING TRANSFER CYCLE"()
   END_RUNG
   RUNG wire#powerrail
      "SUGAR"()
      "RECIPE"()
   END_RUNG
   // the same network as SCL:
   "AUTO SUBOUTPUT"(ENO => #_w1);
   "MFG PROCESS"(EN := #_w1, ENO => #_w2);
   IF #_w2 THEN "MFG TRANSFER CYCLE"(); END_IF;
   "PREMIXING"(ENO => #_w3);
   IF #_w3 THEN "PREMIXING TRANSFER CYCLE"(); END_IF;
   "SUGAR"(ENO => #_w4);
   IF #_w4 THEN "RECIPE"(); END_IF;
END_REGION
END_ORGANIZATION_BLOCK

FUNCTION "AI SCALING" : Void
{ S7_Optimized_Access := 'TRUE' }
VERSION : 0.1

BEGIN
	REGION SYRUP VESSEL TEMP SENSOR
	    "@SCALING AI"("ANALOG INPUT":="SYRUP VESSEL TEMP SENSOR",
	                 "RAW MIN":=0,
	                 "RAW MAX":=27648,
	                 "SCALE MIN":="AI SCALING DB".MIN."SYRUP VESSEL TEMP SENSOR",
	                 "SCALE MAX":="AI SCALING DB".MAX."SYRUP VESSEL TEMP SENSOR",
	                 "PV VALUE"=>"AI SCALING DB".PV."SYRUP VESSEL TEMP SENSOR");
	END_REGION
	
	REGION PREMIXING VESSEL TEMP SENSOR
	    "@SCALING AI"("ANALOG INPUT" := "PREMIXING VESSEL TEMP SENSOR",
	                  "RAW MIN" := 0,
	                  "RAW MAX" := 27648,
	                  "SCALE MIN" := "AI SCALING DB".MIN."PREMIXING VESSEL TEMP SENSOR",
	                  "SCALE MAX" := "AI SCALING DB".MAX."PREMIXING VESSEL TEMP SENSOR",
	                  "PV VALUE" => "AI SCALING DB".PV."PREMIXING VESSEL TEMP SENSOR");
	END_REGION
	
	REGION SUGAR VESSEL TEMP SENSOR
	    "@SCALING AI"("ANALOG INPUT" := "SUGAR VESSEL TEMP SENSOR",
	                  "RAW MIN" := 0,
	                  "RAW MAX" := 27648,
	                  "SCALE MIN" := "AI SCALING DB".MIN."SUGAR VESSEL TEMP SENSOR",
	                  "SCALE MAX" := "AI SCALING DB".MAX."SUGAR VESSEL TEMP SENSOR",
	                  "PV VALUE" => "AI SCALING DB".PV."SUGAR VESSEL TEMP SENSOR");
	END_REGION
	
	REGION STEAM LINE_1 TEMP SENSOR
	    "@SCALING AI"("ANALOG INPUT" := "STEAM LINE_1 TEMP SENSOR",
	                  "RAW MIN" := 0,
	                  "RAW MAX" := 27648,
	                  "SCALE MIN" := "AI SCALING DB".MIN."STEAM LINE_1 TEMP SENSOR",
	                  "SCALE MAX" := "AI SCALING DB".MAX."STEAM LINE_1 TEMP SENSOR",
	                  "PV VALUE" => "AI SCALING DB".PV."STEAM LINE_1 TEMP SENSOR");
	END_REGION
	
	REGION STEAM LINE_2 TEMP SENSOR
	    "@SCALING AI"("ANALOG INPUT" := "STEAM LINE_2 TEMP SENSOR",
	                  "RAW MIN" := 0,
	                  "RAW MAX" := 27648,
	                  "SCALE MIN" := "AI SCALING DB".MIN."STEAM LINE_2 TEMP SENSOR",
	                  "SCALE MAX" := "AI SCALING DB".MAX."STEAM LINE_2 TEMP SENSOR",
	                  "PV VALUE" => "AI SCALING DB".PV."STEAM LINE_2 TEMP SENSOR");
	END_REGION
	
	REGION PRESSURE TRANSMITTER 1
	    "@SCALING AI"("ANALOG INPUT" := "PRESSURE TRANSMITTER 1",
	                  "RAW MIN" := 0,
	                  "RAW MAX" := 27648,
	                  "SCALE MIN" := "AI SCALING DB".MIN."PRESSURE TRANSMITTER 1",
	                  "SCALE MAX" := "AI SCALING DB".MAX."PRESSURE TRANSMITTER 1",
	                  "PV VALUE" => "AI SCALING DB".PV."PRESSURE TRANSMITTER 1");
	END_REGION
	 
	REGION PRESSURE TRANSMITTER 2
	    "@SCALING AI"("ANALOG INPUT" := "PRESSURE TRANSMITTER 2",
	                  "RAW MIN" := 0,
	                  "RAW MAX" := 27648,
	                  "SCALE MIN" := "AI SCALING DB".MIN."PRESSURE TRANSMITTER 2",
	                  "SCALE MAX" := "AI SCALING DB".MAX."PRESSURE TRANSMITTER 2",
	                  "PV VALUE" => "AI SCALING DB".PV."PRESSURE TRANSMITTER 2");
	END_REGION
	
	  REGION VACCIM TRANSMITTER 1
	      "@SCALING AI"("ANALOG INPUT" := "VACCIM TRANSMITTER 1",
	                      "RAW MIN" := 0,
	                      "RAW MAX" := 27648,
	                  "SCALE MIN" := "AI SCALING DB".MIN."VACCIM TRANSMITTER 1",
	                  "SCALE MAX" := "AI SCALING DB".MAX."VACCIM TRANSMITTER 1",
	                  "PV VALUE" => "AI SCALING DB".PV."VACCIM TRANSMITTER 1");
	END_REGION
	
	REGION VACCIM TRANSMITTER 2
	    "@SCALING AI"("ANALOG INPUT" := "VACCIM TRANSMITTER 2",
	                  "RAW MIN" := 0,
	                  "RAW MAX" := 27648,
	                  "SCALE MIN" := "AI SCALING DB".MIN."VACCIM TRANSMITTER 2",
	                  "SCALE MAX" := "AI SCALING DB".MAX."VACCIM TRANSMITTER 2",
	                  "PV VALUE" => "AI SCALING DB".PV."VACCIM TRANSMITTER 2");
	END_REGION
	
	REGION VACCUM TRANSMITTER 3
	    "@SCALING AI"("ANALOG INPUT" := "VACCUM TRANSMITTER 3",
	                  "RAW MIN" := 0,
	                  "RAW MAX" := 27648,
	                  "SCALE MIN" := "AI SCALING DB".MIN."VACCUM TRANSMITTER 3",
	                  "SCALE MAX" := "AI SCALING DB".MAX."VACCUM TRANSMITTER 3",
	                  "PV VALUE" => "AI SCALING DB".PV."VACCUM TRANSMITTER 3");
	END_REGION
	
	REGION SYRUP LOAD CELL
	    "@SCALING AI"("ANALOG INPUT" := "SYRUP LOAD CELL",
	                  "RAW MIN" := 0,
	                  "RAW MAX" := 27648,
	                  "SCALE MIN" := "AI SCALING DB".MIN."SYRUP LOAD CELL",
	                  "SCALE MAX" := "AI SCALING DB".MAX."SYRUP LOAD CELL",
	                  "PV VALUE" => "AI SCALING DB".PV."SYRUP LOAD CELL");
	END_REGION
	
	REGION PREMIXING LOAD CELL
	    "@SCALING AI"("ANALOG INPUT" := "PREMIXING LOAD CELL",
	                  "RAW MIN" := 0,
	                  "RAW MAX" := 27648,
	                  "SCALE MIN" := "AI SCALING DB".MIN."PREMIXING LOAD CELL",
	                  "SCALE MAX" := "AI SCALING DB".MAX."PREMIXING LOAD CELL",
	                  "PV VALUE" => "AI SCALING DB".PV."PREMIXING LOAD CELL");
	END_REGION
	
	REGION SUGAR LOAD CELL
	    "@SCALING AI"("ANALOG INPUT" := "SUGAR LOAD CELL",
	                  "RAW MIN" := 0,
	                  "RAW MAX" := 27648,
	                  "SCALE MIN" := "AI SCALING DB".MIN."SUGAR LOAD CELL",
	                  "SCALE MAX" := "AI SCALING DB".MAX."SUGAR LOAD CELL",
	                  "PV VALUE" => "AI SCALING DB".PV."SUGAR LOAD CELL");
	END_REGION
	
	REGION ULTRASONIC LEVEL SENSOR-1
	    "@SCALING AI"("ANALOG INPUT" := "ULTRASONIC LEVEL SENSOR-1",
	                  "RAW MIN" := 0,
	                  "RAW MAX" := 27648,
	                  "SCALE MIN" := "AI SCALING DB".MIN."ULTRASONIC LEVEL SENSOR-1",
	                  "SCALE MAX" := "AI SCALING DB".MAX."ULTRASONIC LEVEL SENSOR-1",
	                  "PV VALUE" => "AI SCALING DB".PV."ULTRASONIC LEVEL SENSOR-1");
	END_REGION
	
	REGION ULTRASONIC LEVEL SENSOR-2
	    "@SCALING AI"("ANALOG INPUT" := "ULTRASONIC LEVEL SENSOR-2",
	                  "RAW MIN" := 0,
	                  "RAW MAX" := 27648,
	                  "SCALE MIN" := "AI SCALING DB".MIN."ULTRASONIC LEVEL SENSOR-2",
	                  "SCALE MAX" := "AI SCALING DB".MAX."ULTRASONIC LEVEL SENSOR-2",
	                  "PV VALUE" => "AI SCALING DB".PV."ULTRASONIC LEVEL SENSOR-2");
	END_REGION
	
	REGION ULTRASONIC LEVEL SENSOR-3
	    "@SCALING AI"("ANALOG INPUT" := "ULTRASONIC LEVEL SENSOR-3",
	                  "RAW MIN" := 0,
	                  "RAW MAX" := 27648,
	                  "SCALE MIN" := "AI SCALING DB".MIN."ULTRASONIC LEVEL SENSOR-3",
	                  "SCALE MAX" := "AI SCALING DB".MAX."ULTRASONIC LEVEL SENSOR-3",
	                  "PV VALUE" => "AI SCALING DB".PV."ULTRASONIC LEVEL SENSOR-3");
	END_REGION
	
	
	
	
	
	
	
	
	
	
	
	
	
	
END_FUNCTION

FUNCTION "SUBOUTPUT" : Void
{ S7_Optimized_Access := 'TRUE' }
VERSION : 0.1

BEGIN
	REGION SYRUP MFG VESSEL BOTTOM STERROR RUN
	    IF ("MODE SELECTION DB"."MODE BUFF" = 2 AND "MANUAL BIT"."SYRUP MFG VESSEL BOTTOM STERROR RUN")
	        OR ("TRANSFER DB".OUTPUT."SYRUP MFG VESSEL BOTTOM STERROR RUN")
	        OR "AUTO SUBOUTPUT DB"."SYRUP MFG VESSEL BOTTOM STERROR RUN"
	    THEN
	        "DO MAPING"."SYRUP MFG VESSEL BOTTOM STERROR RUN" := TRUE;
	    ELSE
	        "DO MAPING"."SYRUP MFG VESSEL BOTTOM STERROR RUN" := FALSE;
	    END_IF;
	END_REGION
	
	REGION PREMIXING VESSEL BOTTOM STERROR RUN
	    IF ("MODE SELECTION DB"."MODE BUFF" = 2 AND "MANUAL BIT"."PREMIXING VESSEL BOTTOM STERROR RUN")
	        OR ("TRANSFER DB".OUTPUT."PREMIXING VESSEL BOTTOM STERROR RUN")
	        OR "AUTO SUBOUTPUT DB"."PREMIXING VESSEL BOTTOM STERROR RUN"
	    THEN
	        "DO MAPING"."PREMIXING VESSEL BOTTOM STERROR RUN" := TRUE;
	    ELSE
	        "DO MAPING"."PREMIXING VESSEL BOTTOM STERROR RUN" := FALSE;
	    END_IF;
	END_REGION
	
	REGION INLINE 1 HOMOGENIZER MOTOR1 RUN
	    IF ("MODE SELECTION DB"."MODE BUFF" = 2 AND "MANUAL BIT"."INLINE 1 HOMOGENIZER MOTOR1 RUN")
	        OR ("TRANSFER DB".OUTPUT."INLINE 1 HOMOGENIZER MOTOR1 RUN")
	        OR "AUTO SUBOUTPUT DB"."INLINE 1 HOMOGENIZER MOTOR1 RUN"
	    THEN
	        "DO MAPING"."INLINE 1 HOMOGENIZER MOTOR1 RUN" := TRUE;
	    ELSE
	        "DO MAPING"."INLINE 1 HOMOGENIZER MOTOR1 RUN" := FALSE;
	    END_IF;
	END_REGION
	
	REGION INLINE 2 HOMOGENIZER MOTOR 2 RUN
	    IF ("MODE SELECTION DB"."MODE BUFF" = 2 AND "MANUAL BIT"."INLINE 2 HOMOGENIZER MOTOR 2 RUN")
	        OR ("TRANSFER DB".OUTPUT."INLINE 2 HOMOGENIZER MOTOR 2 RUN")
	        OR "AUTO SUBOUTPUT DB"."INLINE 2 HOMOGENIZER MOTOR 2 RUN"
	    THEN
	        "DO MAPING"."INLINE 2 HOMOGENIZER MOTOR 2 RUN" := TRUE;
	    ELSE
	        "DO MAPING"."INLINE 2 HOMOGENIZER MOTOR 2 RUN" := FALSE;
	    END_IF;
	END_REGION
	
	REGION FILTER PRESS MOTOR 1 RUN
	    IF ("MODE SELECTION DB"."MODE BUFF" = 2 AND "MANUAL BIT"."FILTER PRESS MOTOR 1 RUN")
	        OR ("TRANSFER DB".OUTPUT."FILTER PRESS MOTOR 1 RUN")
	        OR "AUTO SUBOUTPUT DB"."FILTER PRESS MOTOR 1 RUN"
	    THEN
	        "DO MAPING"."FILTER PRESS MOTOR 1 RUN" := TRUE;
	    ELSE
	        "DO MAPING"."FILTER PRESS MOTOR 1 RUN" := FALSE;
	    END_IF;
	END_REGION
	
	REGION FILTER PRESS MOTOR 2 RUN
	    IF ("MODE SELECTION DB"."MODE BUFF" = 2 AND "MANUAL BIT"."FILTER PRESS MOTOR 2 RUN")
	        OR ("TRANSFER DB".OUTPUT."FILTER PRESS MOTOR 2 RUN")
	        OR "AUTO SUBOUTPUT DB"."FILTER PRESS MOTOR 2 RUN"
	    THEN
	        "DO MAPING"."FILTER PRESS MOTOR 2 RUN" := TRUE;
	    ELSE
	        "DO MAPING"."FILTER PRESS MOTOR 2 RUN" := FALSE;
	    END_IF;
	END_REGION
	
	REGION VACCUM PUMP MOTOR-W 1 RUN
	    IF ("MODE SELECTION DB"."MODE BUFF" = 2 AND "MANUAL BIT"."VACCUM PUMP MOTOR-W 1 RUN" OR "MANUAL BIT"."VACCUM PUMP MOTOR-W 1 RUN_1")
	        OR "AUTO SUBOUTPUT DB"."VACCUM PUMP MOTOR-W 1 RUN"
	    THEN
	        "DO MAPING"."VACCUM PUMP MOTOR-W 1 RUN" := TRUE;
	    ELSE
	        "DO MAPING"."VACCUM PUMP MOTOR-W 1 RUN" := FALSE;
	    END_IF;
	END_REGION
	
	REGION VACCUMP PUMP MOTOR-S2 RUN
	    IF ("MODE SELECTION DB"."MODE BUFF" = 2 AND "MANUAL BIT"."VACCUMP PUMP MOTOR-S2 RUN" OR "MANUAL BIT"."VACCUMP PUMP MOTOR-S2 RUN_1")
	        
	        OR "AUTO SUBOUTPUT DB"."VACCUMP PUMP MOTOR-S2 RUN"
	    THEN
	        "DO MAPING"."VACCUMP PUMP MOTOR-S2 RUN" := TRUE;
	    ELSE
	        "DO MAPING"."VACCUMP PUMP MOTOR-S2 RUN" := FALSE;
	    END_IF;
	END_REGION
	
	REGION VACCUMP PUMP MOTOR-W 3 RUN
	    IF ("MODE SELECTION DB"."MODE BUFF" = 2 AND "MANUAL BIT"."VACCUMP PUMP MOTOR-W 3 RUN")
	        OR "AUTO SUBOUTPUT DB"."VACCUMP PUMP MOTOR-W 3 RUN"
	    THEN
	        "DO MAPING"."VACCUMP PUMP MOTOR-W 3 RUN" := TRUE;
	    ELSE
	        "DO MAPING"."VACCUMP PUMP MOTOR-W 3 RUN" := FALSE;
	    END_IF;
	END_REGION
	
	REGION VACCUMP PUMP MOTOR-S 4 RUN
	    IF ("MODE SELECTION DB"."MODE BUFF" = 2 AND "MANUAL BIT"."VACCUMP PUMP MOTOR-S 4 RUN")
	        OR "AUTO SUBOUTPUT DB"."VACCUMP PUMP MOTOR-S 4 RUN"
	    THEN
	        "DO MAPING"."VACCUMP PUMP MOTOR-S 4 RUN" := TRUE;
	    ELSE
	        "DO MAPING"."VACCUMP PUMP MOTOR-S 4 RUN" := FALSE;
	    END_IF;
	END_REGION
	
	REGION SUGAR VESSEL BOTTOM STERROR RUN
	    IF ("MODE SELECTION DB"."MODE BUFF" = 2 AND "MANUAL BIT"."SUGAR VESSEL BOTTOM STERROR RUN")
	        OR ("TRANSFER DB".OUTPUT."SUGAR VESSEL BOTTOM STERROR RUN")
	        OR "AUTO SUBOUTPUT DB"."SUGAR VESSEL BOTTOM STERROR RUN"
	    THEN
	        "DO MAPING"."SUGAR VESSEL BOTTOM STERROR RUN" := TRUE;
	    ELSE
	        "DO MAPING"."SUGAR VESSEL BOTTOM STERROR RUN" := FALSE;
	    END_IF;
	END_REGION
	
	REGION BASKET FILTER MOTOR RUN
	    IF ("MODE SELECTION DB"."MODE BUFF" = 2 AND "MANUAL BIT"."BASKET FILTER MOTOR RUN")
	        OR ("TRANSFER DB".OUTPUT."BASKET FILTER MOTOR RUN")
	        OR "AUTO SUBOUTPUT DB"."BASKET FILTER MOTOR RUN"
	    THEN
	        "DO MAPING"."BASKET FILTER MOTOR RUN" := TRUE;
	    ELSE
	        "DO MAPING"."BASKET FILTER MOTOR RUN" := FALSE;
	    END_IF;
	END_REGION
	
	REGION PBV-01 INGREDIENT INLET
	    IF ("MODE SELECTION DB"."MODE BUFF" = 2 AND "MANUAL BIT"."PBV-01 INGREDIENT INLET")
	        OR ("TRANSFER DB".OUTPUT."PBV-01 INGREDIENT INLET")
	        OR "AUTO SUBOUTPUT DB"."PBV-01 INGREDIENT INLET"
	    THEN
	        "DO MAPING"."PBV-01 INGREDIENT INLET" := TRUE;
	    ELSE
	        "DO MAPING"."PBV-01 INGREDIENT INLET" := FALSE;
	    END_IF;
	END_REGION
	
	REGION PBV-02 CIP INLET (SPRAY BALL)
	    IF ("MODE SELECTION DB"."MODE BUFF" = 2 AND "MANUAL BIT"."PBV-02 CIP INLET (SPRAY BALL)")
	        OR ("TRANSFER DB".OUTPUT."PBV-02 CIP INLET (SPRAY BALL)")
	        OR "AUTO SUBOUTPUT DB"."PBV-02 CIP INLET (SPRAY BALL)"
	    THEN
	        "DO MAPING"."PBV-02 CIP INLET (SPRAY BALL)" := TRUE;
	    ELSE
	        "DO MAPING"."PBV-02 CIP INLET (SPRAY BALL)" := FALSE;
	    END_IF;
	END_REGION
	
	REGION PBV-03 VENT FILTER ISOLATION
	    IF ("MODE SELECTION DB"."MODE BUFF" = 2 AND "MANUAL BIT"."PBV-03 VENT FILTER ISOLATION")
	        OR ("TRANSFER DB".OUTPUT."PBV-03 VENT FILTER ISOLATION")
	        OR "AUTO SUBOUTPUT DB"."PBV-03 VENT FILTER ISOLATION"
	    THEN
	        "DO MAPING"."PBV-03 VENT FILTER ISOLATION" := TRUE;
	    ELSE
	        "DO MAPING"."PBV-03 VENT FILTER ISOLATION" := FALSE;
	    END_IF;
	END_REGION
	
	REGION PBV-04 PW INLET
	    IF ("MODE SELECTION DB"."MODE BUFF" = 2 AND "MANUAL BIT"."PBV-04 PW INLET")
	        OR ("TRANSFER DB".OUTPUT."PBV-04 PW INLET")
	        OR "AUTO SUBOUTPUT DB"."PBV-04 PW INLET"
	    THEN
	        "DO MAPING"."PBV-04 PW INLET" := TRUE;
	    ELSE
	        "DO MAPING"."PBV-04 PW INLET" := FALSE;
	    END_IF;
	END_REGION
	
	REGION PBV-07 PREMIX TANK DRAIN VALVE
	    IF ("MODE SELECTION DB"."MODE BUFF" = 2 AND "MANUAL BIT"."PBV-07 PREMIX TANK DRAIN VALVE")
	        OR ("TRANSFER DB".OUTPUT."PBV-07 PREMIX TANK DRAIN VALVE")
	        OR "AUTO SUBOUTPUT DB"."PBV-07 PREMIX TANK DRAIN VALVE"
	    THEN
	        "DO MAPING"."PBV-07 PREMIX TANK DRAIN VALVE" := TRUE;
	    ELSE
	        "DO MAPING"."PBV-07 PREMIX TANK DRAIN VALVE" := FALSE;
	    END_IF;
	END_REGION
	
	REGION PAV-09 JACKET STEAM INLET
	    IF ("MODE SELECTION DB"."MODE BUFF" = 2 AND "MANUAL BIT"."PAV-09 JACKET STEAM INLET"
	        AND NOT "DO MAPING"."PAV-13 WATER COOLING INLET" AND "LEVEL BUFF".PREMIXING_TEMP<>1)
	        OR ("TRANSFER DB".OUTPUT."PAV-09 JACKET STEAM INLET")
	        OR "AUTO SUBOUTPUT DB"."PAV-09 JACKET STEAM INLET"
	    THEN
	        "DO MAPING"."PAV-09 JACKET STEAM INLET" := TRUE;
	    ELSE
	        "DO MAPING"."PAV-09 JACKET STEAM INLET" := FALSE;
	    END_IF;
	END_REGION
	
	REGION PAV-10 JACKET CONDENSATE DRAIN
	    IF ("MODE SELECTION DB"."MODE BUFF" = 2 AND "MANUAL BIT"."PAV-10 JACKET CONDENSATE DRAIN"
	        AND NOT "DO MAPING"."PAV-13 WATER COOLING INLET" AND "LEVEL BUFF".PREMIXING_TEMP<>1)
	        OR ("TRANSFER DB".OUTPUT."PAV-10 JACKET CONDENSATE DRAIN")
	        OR "AUTO SUBOUTPUT DB"."PAV-10 JACKET CONDENSATE DRAIN"
	    THEN
	        "DO MAPING"."PAV-10 JACKET CONDENSATE DRAIN" := TRUE;
	    ELSE
	        "DO MAPING"."PAV-10 JACKET CONDENSATE DRAIN" := FALSE;
	    END_IF;
	END_REGION
	
	REGION PAV-11 JACKET BYPASS DRAIN VALVE
	    IF ("MODE SELECTION DB"."MODE BUFF" = 2 AND "MANUAL BIT"."PAV-11 JACKET BYPASS DRAIN VALVE")
	        OR ("TRANSFER DB".OUTPUT."PAV-11 JACKET BYPASS DRAIN VALVE")
	        OR "AUTO SUBOUTPUT DB"."PAV-11 JACKET BYPASS DRAIN VALVE"
	    THEN
	        "DO MAPING"."PAV-11 JACKET BYPASS DRAIN VALVE" := TRUE;
	    ELSE
	        "DO MAPING"."PAV-11 JACKET BYPASS DRAIN VALVE" := FALSE;
	    END_IF;
	END_REGION
	
	REGION PAV-12 SEAL COOLING INLET
	    IF ("MODE SELECTION DB"."MODE BUFF" = 2 AND "MANUAL BIT"."PAV-12 SEAL COOLING INLET")
	        OR ("TRANSFER DB".OUTPUT."PAV-12 SEAL COOLING INLET")
	        OR "AUTO SUBOUTPUT DB"."PAV-12 SEAL COOLING INLET"
	    THEN
	        "DO MAPING"."PAV-12 SEAL COOLING INLET" := TRUE;
	    ELSE
	        "DO MAPING"."PAV-12 SEAL COOLING INLET" := FALSE;
	    END_IF;
	END_REGION
	
	REGION PAV-13 WATER COOLING INLET
	    IF ("MODE SELECTION DB"."MODE BUFF" = 2 AND "MANUAL BIT"."PAV-13 WATER COOLING INLET" AND NOT "DO MAPING"."PAV-09 JACKET STEAM INLET")
	        OR ("TRANSFER DB".OUTPUT."PAV-13 WATER COOLING INLET")
	        OR "AUTO SUBOUTPUT DB"."PAV-13 WATER COOLING INLET"
	    THEN
	        "DO MAPING"."PAV-13 WATER COOLING INLET" := TRUE;
	    ELSE
	        "DO MAPING"."PAV-13 WATER COOLING INLET" := FALSE;
	    END_IF;
	END_REGION
	
	REGION PAV-14 WATER COOLING OUTLET
	    IF ("MODE SELECTION DB"."MODE BUFF" = 2 AND "MANUAL BIT"."PAV-14 WATER COOLING OUTLET")
	        OR ("TRANSFER DB".OUTPUT."PAV-14 WATER COOLING OUTLET")
	        OR "AUTO SUBOUTPUT DB"."PAV-14 WATER COOLING OUTLET"
	    THEN
	        "DO MAPING"."PAV-14 WATER COOLING OUTLET" := TRUE;
	    ELSE
	        "DO MAPING"."PAV-14 WATER COOLING OUTLET" := FALSE;
	    END_IF;
	END_REGION
	
	REGION PBV-15 VACUUM INLET
	    IF ("MODE SELECTION DB"."MODE BUFF" = 2 AND "MANUAL BIT"."PBV-15 VACUUM INLET")
	        OR ("TRANSFER DB".OUTPUT."PBV-15 VACUUM INLET")
	        OR "AUTO SUBOUTPUT DB"."PBV-15 VACUUM INLET"
	    THEN
	        "DO MAPING"."PBV-15 VACUUM INLET" := TRUE;
	    ELSE
	        "DO MAPING"."PBV-15 VACUUM INLET" := FALSE;
	    END_IF;
	END_REGION
	
	REGION PBV-16 VACUUM VENT VALVE
	    IF ("MODE SELECTION DB"."MODE BUFF" = 2 AND "MANUAL BIT"."PBV-16 VACUUM VENT VALVE")
	        OR ("TRANSFER DB".OUTPUT."PBV-16 VACUUM VENT VALVE")
	        OR "AUTO SUBOUTPUT DB"."PBV-16 VACUUM VENT VALVE"
	    THEN
	        "DO MAPING"."PBV-16 VACUUM VENT VALVE" := TRUE;
	    ELSE
	        "DO MAPING"."PBV-16 VACUUM VENT VALVE" := FALSE;
	    END_IF;
	END_REGION
	
	REGION PFBV-17 TANK OUTLET VALVE
	    IF ("MODE SELECTION DB"."MODE BUFF" = 2 AND "MANUAL BIT"."PFBV-17 TANK OUTLET VALVE")
	        OR ("TRANSFER DB".OUTPUT."PFBV-17 TANK OUTLET VALVE")
	        OR "AUTO SUBOUTPUT DB"."PFBV-17 TANK OUTLET VALVE"
	    THEN
	        "DO MAPING"."PFBV-17 TANK OUTLET VALVE" := TRUE;
	    ELSE
	        "DO MAPING"."PFBV-17 TANK OUTLET VALVE" := FALSE;
	    END_IF;
	END_REGION
	
	REGION PBV-19 PW INLET
	    IF ("MODE SELECTION DB"."MODE BUFF" = 2 AND "MANUAL BIT"."PBV-19 PW INLET")
	        OR ("TRANSFER DB".OUTPUT."PBV-19 PW INLET")
	        OR "AUTO SUBOUTPUT DB"."PBV-19 PW INLET"
	    THEN
	        "DO MAPING"."PBV-19 PW INLET" := TRUE;
	    ELSE
	        "DO MAPING"."PBV-19 PW INLET" := FALSE;
	    END_IF;
	END_REGION
	
	REGION PBV-20 CIP INLET (SPRAY BALL)
	    IF ("MODE SELECTION DB"."MODE BUFF" = 2 AND "MANUAL BIT"."PBV-20 CIP INLET (SPRAY BALL)")
	        OR ("TRANSFER DB".OUTPUT."PBV-20 CIP INLET (SPRAY BALL)")
	        OR "AUTO SUBOUTPUT DB"."PBV-20 CIP INLET (SPRAY BALL)"
	    THEN
	        "DO MAPING"."PBV-20 CIP INLET (SPRAY BALL)" := TRUE;
	    ELSE
	        "DO MAPING"."PBV-20 CIP INLET (SPRAY BALL)" := FALSE;
	    END_IF;
	END_REGION
	
	REGION PBV-21 VENT FILTER ISOLATION
	    IF ("MODE SELECTION DB"."MODE BUFF" = 2 AND "MANUAL BIT"."PBV-21 VENT FILTER ISOLATION")
	        OR ("TRANSFER DB".OUTPUT."PBV-21 VENT FILTER ISOLATION")
	        OR "AUTO SUBOUTPUT DB"."PBV-21 VENT FILTER ISOLATION"
	    THEN
	        "DO MAPING"."PBV-21 VENT FILTER ISOLATION" := TRUE;
	    ELSE
	        "DO MAPING"."PBV-21 VENT FILTER ISOLATION" := FALSE;
	    END_IF;
	END_REGION
	
	REGION PBV-22 INGREDIENT INLET (SUGAR INLET)
	    IF ("MODE SELECTION DB"."MODE BUFF" = 2 AND "MANUAL BIT"."PBV-22 INGREDIENT INLET (SUGAR INLET)")
	        OR ("TRANSFER DB".OUTPUT."PBV-22 INGREDIENT INLET (SUGAR INLET)")
	        OR "AUTO SUBOUTPUT DB"."PBV-22 INGREDIENT INLET (SUGAR INLET)"
	    THEN
	        "DO MAPING"."PBV-22 INGREDIENT INLET (SUGAR INLET)" := TRUE;
	    ELSE
	        "DO MAPING"."PBV-22 INGREDIENT INLET (SUGAR INLET)" := FALSE;
	    END_IF;
	END_REGION
	
	REGION PBV-25 BOTTOM OUTLET TO DRAIN VALVE
	    IF ("MODE SELECTION DB"."MODE BUFF" = 2 AND "MANUAL BIT"."PBV-25 BOTTOM OUTLET TO DRAIN VALVE")
	        OR ("TRANSFER DB".OUTPUT."PBV-25 BOTTOM OUTLET TO DRAIN VALVE")
	        OR "AUTO SUBOUTPUT DB"."PBV-25 BOTTOM OUTLET TO DRAIN VALVE"
	    THEN
	        "DO MAPING"."PBV-25 BOTTOM OUTLET TO DRAIN VALVE" := TRUE;
	    ELSE
	        "DO MAPING"."PBV-25 BOTTOM OUTLET TO DRAIN VALVE" := FALSE;
	    END_IF;
	END_REGION
	
	REGION PAV-27 JACKET STEAM INLET
	    IF ("MODE SELECTION DB"."MODE BUFF" = 2 AND "MANUAL BIT"."PAV-27 JACKET STEAM INLET" AND "LEVEL BUFF".SUGAR_TEMP<>1)
	        OR ("TRANSFER DB".OUTPUT."PAV-27 JACKET STEAM INLET")
	        OR "AUTO SUBOUTPUT DB"."PAV-27 JACKET STEAM INLET"
	    THEN
	        "DO MAPING"."PAV-27 JACKET STEAM INLET" := TRUE;
	    ELSE
	        "DO MAPING"."PAV-27 JACKET STEAM INLET" := FALSE;
	    END_IF;
	END_REGION
	
	REGION PAV-28 SEAL COOLING INLET
	    IF ("MODE SELECTION DB"."MODE BUFF" = 2 AND "MANUAL BIT"."PAV-28 SEAL COOLING INLET")
	        OR ("TRANSFER DB".OUTPUT."PAV-28 SEAL COOLING INLET")
	        OR "AUTO SUBOUTPUT DB"."PAV-28 SEAL COOLING INLET"
	    THEN
	        "DO MAPING"."PAV-28 SEAL COOLING INLET" := TRUE;
	    ELSE
	        "DO MAPING"."PAV-28 SEAL COOLING INLET" := FALSE;
	    END_IF;
	END_REGION
	
	REGION PAV-29 JACKET CONDENSATE DRAIN
	    IF ("MODE SELECTION DB"."MODE BUFF" = 2 AND "MANUAL BIT"."PAV-29 JACKET CONDENSATE DRAIN")
	        OR ("TRANSFER DB".OUTPUT."PAV-29 JACKET CONDENSATE DRAIN")
	        OR "AUTO SUBOUTPUT DB"."PAV-29 JACKET CONDENSATE DRAIN"
	    THEN
	        "DO MAPING"."PAV-29 JACKET CONDENSATE DRAIN" := TRUE;
	    ELSE
	        "DO MAPING"."PAV-29 JACKET CONDENSATE DRAIN" := FALSE;
	    END_IF;
	END_REGION
	
	REGION PBV-30 VACUUM INLET VALVE
	    IF ("MODE SELECTION DB"."MODE BUFF" = 2 AND "MANUAL BIT"."PBV-30 VACUUM INLET VALVE")
	        OR ("TRANSFER DB".OUTPUT."PBV-30 VACUUM INLET VALVE")
	        OR "AUTO SUBOUTPUT DB"."PBV-30 VACUUM INLET VALVE"
	    THEN
	        "DO MAPING"."PBV-30 VACUUM INLET VALVE" := TRUE;
	    ELSE
	        "DO MAPING"."PBV-30 VACUUM INLET VALVE" := FALSE;
	    END_IF;
	END_REGION
	
	REGION PBV-31 VACUUM VENT VALVE
	    IF ("MODE SELECTION DB"."MODE BUFF" = 2 AND "MANUAL BIT"."PBV-31 VACUUM VENT VALVE")
	        OR ("TRANSFER DB".OUTPUT."PBV-31 VACUUM VENT VALVE")
	        OR "AUTO SUBOUTPUT DB"."PBV-31 VACUUM VENT VALVE"
	    THEN
	        "DO MAPING"."PBV-31 VACUUM VENT VALVE" := TRUE;
	    ELSE
	        "DO MAPING"."PBV-31 VACUUM VENT VALVE" := FALSE;
	    END_IF;
	END_REGION
	
	REGION PFBV-32 TANK OUTLET VALVE
	    IF ("MODE SELECTION DB"."MODE BUFF" = 2 AND "MANUAL BIT"."PFBV-32 TANK OUTLET VALVE")
	        OR ("TRANSFER DB".OUTPUT."PFBV-32 TANK OUTLET VALVE")
	        OR "AUTO SUBOUTPUT DB"."PFBV-32 TANK OUTLET VALVE"
	    THEN
	        "DO MAPING"."PFBV-32 TANK OUTLET VALVE" := TRUE;
	    ELSE
	        "DO MAPING"."PFBV-32 TANK OUTLET VALVE" := FALSE;
	    END_IF;
	END_REGION
	
	REGION PBV-36 PW INLET
	    IF ("MODE SELECTION DB"."MODE BUFF" = 2 AND "MANUAL BIT"."PBV-36 PW INLET")
	        OR ("TRANSFER DB".OUTPUT."PBV-36 PW INLET")
	        OR "AUTO SUBOUTPUT DB"."PBV-36 PW INLET"
	    THEN
	        "DO MAPING"."PBV-36 PW INLET" := TRUE;
	    ELSE
	        "DO MAPING"."PBV-36 PW INLET" := FALSE;
	    END_IF;
	END_REGION
	
	REGION PBV-37 VENT FILTER ISOLATION
	    IF ("MODE SELECTION DB"."MODE BUFF" = 2 AND "MANUAL BIT"."PBV-37 VENT FILTER ISOLATION")
	        OR ("TRANSFER DB".OUTPUT."PBV-37 VENT FILTER ISOLATION")
	        OR "AUTO SUBOUTPUT DB"."PBV-37 VENT FILTER ISOLATION"
	    THEN
	        "DO MAPING"."PBV-37 VENT FILTER ISOLATION" := TRUE;
	    ELSE
	        "DO MAPING"."PBV-37 VENT FILTER ISOLATION" := FALSE;
	    END_IF;
	END_REGION
	
	REGION PBV-38 CIP INLET LINE
	    IF ("MODE SELECTION DB"."MODE BUFF" = 2 AND "MANUAL BIT"."PBV-38 CIP INLET LINE")
	        OR ("TRANSFER DB".OUTPUT."PBV-38 CIP INLET LINE")
	        OR "AUTO SUBOUTPUT DB"."PBV-38 CIP INLET LINE"
	    THEN
	        "DO MAPING"."PBV-38 CIP INLET LINE" := TRUE;
	    ELSE
	        "DO MAPING"."PBV-38 CIP INLET LINE" := FALSE;
	    END_IF;
	END_REGION
	
	REGION PBV-41 MFG TANK DRAIN VALVE
	    IF ("MODE SELECTION DB"."MODE BUFF" = 2 AND "MANUAL BIT"."PBV-41 MFG TANK DRAIN VALVE")
	        OR ("TRANSFER DB".OUTPUT."PBV-41 MFG TANK DRAIN VALVE")
	        OR "AUTO SUBOUTPUT DB"."PBV-41 MFG TANK DRAIN VALVE"
	    THEN
	        "DO MAPING"."PBV-41 MFG TANK DRAIN VALVE" := TRUE;
	    ELSE
	        "DO MAPING"."PBV-41 MFG TANK DRAIN VALVE" := FALSE;
	    END_IF;
	END_REGION
	
	REGION PAV-50 JACKET STEAM INLET
	    IF ("MODE SELECTION DB"."MODE BUFF" = 2 AND "MANUAL BIT"."PAV-50 JACKET STEAM INLET"
	        AND NOT "DO MAPING"."PAV-52 WATER COOLING INLET" AND "LEVEL BUFF"."SYRUP MFG_TEMP"<>1)
	        OR ("TRANSFER DB".OUTPUT."PAV-50 JACKET STEAM INLET")
	        OR "AUTO SUBOUTPUT DB"."PAV-50 JACKET STEAM INLET"
	    THEN
	        "DO MAPING"."PAV-50 JACKET STEAM INLET" := TRUE;
	    ELSE
	        "DO MAPING"."PAV-50 JACKET STEAM INLET" := FALSE;
	    END_IF;
	END_REGION
	
	REGION PAV-51 WATER COOLING OUTLET
	    IF ("MODE SELECTION DB"."MODE BUFF" = 2 AND "MANUAL BIT"."PAV-51 WATER COOLING OUTLET"
	        AND NOT "DO MAPING"."PAV-54 JACKET STEAM OUTLET VALVE")
	        OR ("TRANSFER DB".OUTPUT."PAV-51 WATER COOLING OUTLET")
	        OR "AUTO SUBOUTPUT DB"."PAV-51 WATER COOLING OUTLET"
	    THEN
	        "DO MAPING"."PAV-51 WATER COOLING OUTLET" := TRUE;
	    ELSE
	        "DO MAPING"."PAV-51 WATER COOLING OUTLET" := FALSE;
	    END_IF;
	END_REGION
	
	REGION PAV-52 WATER COOLING INLET
	    IF ("MODE SELECTION DB"."MODE BUFF" = 2 AND "MANUAL BIT"."PAV-52 WATER COOLING INLET"
	        AND NOT "DO MAPING"."PAV-54 JACKET STEAM OUTLET VALVE")
	        OR ("TRANSFER DB".OUTPUT."PAV-52 WATER COOLING INLET")
	        OR "AUTO SUBOUTPUT DB"."PAV-52 WATER COOLING INLET"
	    THEN
	        "DO MAPING"."PAV-52 WATER COOLING INLET" := TRUE;
	    ELSE
	        "DO MAPING"."PAV-52 WATER COOLING INLET" := FALSE;
	    END_IF;
	END_REGION
	
	REGION PAV-53 SEAL COOLING INLET
	    IF ("MODE SELECTION DB"."MODE BUFF" = 2 AND "MANUAL BIT"."PAV-53 SEAL COOLING INLET")
	        OR ("TRANSFER DB".OUTPUT."PAV-53 SEAL COOLING INLET")
	        OR "AUTO SUBOUTPUT DB"."PAV-53 SEAL COOLING INLET"
	    THEN
	        "DO MAPING"."PAV-53 SEAL COOLING INLET" := TRUE;
	    ELSE
	        "DO MAPING"."PAV-53 SEAL COOLING INLET" := FALSE;
	    END_IF;
	END_REGION
	
	REGION PAV-54 JACKET STEAM OUTLET VALVE
	    IF ("MODE SELECTION DB"."MODE BUFF" = 2 AND "MANUAL BIT"."PAV-54 JACKET STEAM OUTLET VALVE"
	        AND NOT "DO MAPING"."PAV-52 WATER COOLING INLET" AND "LEVEL BUFF"."SYRUP MFG_TEMP"<>1)
	        OR ("TRANSFER DB".OUTPUT."PAV-54 JACKET STEAM OUTLET VALVE")
	        OR "AUTO SUBOUTPUT DB"."PAV-54 JACKET STEAM OUTLET VALVE"
	    THEN
	        "DO MAPING"."PAV-54 JACKET STEAM OUTLET VALVE" := TRUE;
	    ELSE
	        "DO MAPING"."PAV-54 JACKET STEAM OUTLET VALVE" := FALSE;
	    END_IF;
	END_REGION
	
	REGION PAV-55 JACKET CONDENSATE BYPASS DRAIN
	    IF ("MODE SELECTION DB"."MODE BUFF" = 2 AND "MANUAL BIT"."PAV-55 JACKET CONDENSATE BYPASS DRAIN")
	        OR ("TRANSFER DB".OUTPUT."PAV-55 JACKET CONDENSATE BYPASS DRAIN")
	        OR "AUTO SUBOUTPUT DB"."PAV-55 JACKET CONDENSATE BYPASS DRAIN"
	    THEN
	        "DO MAPING"."PAV-55 JACKET CONDENSATE BYPASS DRAIN" := TRUE;
	    ELSE
	        "DO MAPING"."PAV-55 JACKET CONDENSATE BYPASS DRAIN" := FALSE;
	    END_IF;
	END_REGION
	
	REGION PAV-56 INLINE HOMO. SEAL COOLING INLET
	    IF ("MODE SELECTION DB"."MODE BUFF" = 2 AND "MANUAL BIT"."PAV-56 INLINE HOMO. SEAL COOLING INLET")
	        OR ("TRANSFER DB".OUTPUT."PAV-56 INLINE HOMO. SEAL COOLING INLET")
	        OR "AUTO SUBOUTPUT DB"."PAV-56 INLINE HOMO. SEAL COOLING INLET"
	    THEN
	        "DO MAPING"."PAV-56 INLINE HOMO. SEAL COOLING INLET" := TRUE;
	    ELSE
	        "DO MAPING"."PAV-56 INLINE HOMO. SEAL COOLING INLET" := FALSE;
	    END_IF;
	END_REGION
	
	REGION PBV-57 VACUUM INLET VALVE
	    IF ("MODE SELECTION DB"."MODE BUFF" = 2 AND "MANUAL BIT"."PBV-57 VACUUM INLET VALVE")
	        OR ("TRANSFER DB".OUTPUT."PBV-57 VACUUM INLET VALVE")
	        OR "AUTO SUBOUTPUT DB"."PBV-57 VACUUM INLET VALVE"
	    THEN
	        "DO MAPING"."PBV-57 VACUUM INLET VALVE" := TRUE;
	    ELSE
	        "DO MAPING"."PBV-57 VACUUM INLET VALVE" := FALSE;
	    END_IF;
	END_REGION
	
	REGION PFBV-59 TANK OUTLET VALVE
	    IF ("MODE SELECTION DB"."MODE BUFF" = 2 AND "MANUAL BIT"."PFBV-59 TANK OUTLET VALVE")
	        OR ("TRANSFER DB".OUTPUT."PFBV-59 TANK OUTLET VALVE")
	        OR "AUTO SUBOUTPUT DB"."PFBV-59 TANK OUTLET VALVE"
	    THEN
	        "DO MAPING"."PFBV-59 TANK OUTLET VALVE" := TRUE;
	    ELSE
	        "DO MAPING"."PFBV-59 TANK OUTLET VALVE" := FALSE;
	    END_IF;
	END_REGION
	
	REGION PBV-79 BASKET FILTER INLET
	    IF ("MODE SELECTION DB"."MODE BUFF" = 2 AND "MANUAL BIT"."PBV-79 BASKET FILTER INLET")
	        OR ("TRANSFER DB".OUTPUT."PBV-79 BASKET FILTER INLET")
	        OR "AUTO SUBOUTPUT DB"."PBV-79 BASKET FILTER INLET"
	    THEN
	        "DO MAPING"."PBV-79 BASKET FILTER INLET" := TRUE;
	    ELSE
	        "DO MAPING"."PBV-79 BASKET FILTER INLET" := FALSE;
	    END_IF;
	END_REGION
	
	REGION PBV-80 BOTTOM OUTLET TO BASKET FILTER
	    IF ("MODE SELECTION DB"."MODE BUFF" = 2 AND "MANUAL BIT"."PBV-80 BOTTOM OUTLET TO BASKET FILTER")
	        OR ("TRANSFER DB".OUTPUT."PBV-80 BOTTOM OUTLET TO BASKET FILTER")
	        OR "AUTO SUBOUTPUT DB"."PBV-80 BOTTOM OUTLET TO BASKET FILTER"
	    THEN
	        "DO MAPING"."PBV-80 BOTTOM OUTLET TO BASKET FILTER" := TRUE;
	    ELSE
	        "DO MAPING"."PBV-80 BOTTOM OUTLET TO BASKET FILTER" := FALSE;
	    END_IF;
	END_REGION
	
	REGION PBV-81 TANK BOTTOM OUTLET TO CIP OUTLET
	    IF ("MODE SELECTION DB"."MODE BUFF" = 2 AND "MANUAL BIT"."PBV-81 TANK BOTTOM OUTLET TO CIP OUTLET")
	        OR ("TRANSFER DB".OUTPUT."PBV-81 TANK BOTTOM OUTLET TO CIP OUTLET")
	        OR "AUTO SUBOUTPUT DB"."PBV-81 TANK BOTTOM OUTLET TO CIP OUTLET"
	    THEN
	        "DO MAPING"."PBV-81 TANK BOTTOM OUTLET TO CIP OUTLET" := TRUE;
	    ELSE
	        "DO MAPING"."PBV-81 TANK BOTTOM OUTLET TO CIP OUTLET" := FALSE;
	    END_IF;
	END_REGION
	
	REGION PBV-82 CIP ISOLATION
	    IF ("MODE SELECTION DB"."MODE BUFF" = 2 AND "MANUAL BIT"."PBV-82 CIP ISOLATION")
	        OR ("TRANSFER DB".OUTPUT."PBV-82 CIP ISOLATION")
	        OR "AUTO SUBOUTPUT DB"."PBV-82 CIP ISOLATION"
	    THEN
	        "DO MAPING"."PBV-82 CIP ISOLATION" := TRUE;
	    ELSE
	        "DO MAPING"."PBV-82 CIP ISOLATION" := FALSE;
	    END_IF;
	END_REGION
	
	REGION PBV-83 PREMIX TRANSFER TO MFG VESSEL TRANSFER
	    IF ("MODE SELECTION DB"."MODE BUFF" = 2 AND "MANUAL BIT"."PBV-83 PREMIX TRANSFER TO MFG VESSEL TRANSFER (TOP DISH)")
	        OR ("TRANSFER DB".OUTPUT."PBV-83 PREMIX TRANSFER TO MFG VESSEL TRANSFER (TOP DISH)")
	        OR "AUTO SUBOUTPUT DB"."PBV-83 PREMIX TRANSFER TO MFG VESSEL TRANSFER (TOP DISH)"
	    THEN
	        "DO MAPING"."PBV-83 PREMIX TRANSFER TO MFG VESSEL TRANSFER (TOP DISH)" := TRUE;
	    ELSE
	        "DO MAPING"."PBV-83 PREMIX TRANSFER TO MFG VESSEL TRANSFER (TOP DISH)" := FALSE;
	    END_IF;
	END_REGION
	
	REGION PBV-84 FROM TANK OUTLET TO CIP OUTLET
	    IF ("MODE SELECTION DB"."MODE BUFF" = 2 AND "MANUAL BIT"."PBV-84 FROM TANK OUTLET TO CIP OUTLET")
	        OR ("TRANSFER DB".OUTPUT."PBV-84 FROM TANK OUTLET TO CIP OUTLET")
	        OR "AUTO SUBOUTPUT DB"."PBV-84 FROM TANK OUTLET TO CIP OUTLET"
	    THEN
	        "DO MAPING"."PBV-84 FROM TANK OUTLET TO CIP OUTLET" := TRUE;
	    ELSE
	        "DO MAPING"."PBV-84 FROM TANK OUTLET TO CIP OUTLET" := FALSE;
	    END_IF;
	END_REGION
	
	REGION PBV-85 SORBITOL INLET LINE
	    IF ("MODE SELECTION DB"."MODE BUFF" = 2 AND "MANUAL BIT"."PBV-85 SORBITOL INLET LINE")
	        OR ("TRANSFER DB".OUTPUT."PBV-85 SORBITOL INLET LINE")
	        OR "AUTO SUBOUTPUT DB"."PBV-85 SORBITOL INLET LINE"
	    THEN
	        "DO MAPING"."PBV-85 SORBITOL INLET LINE" := TRUE;
	    ELSE
	        "DO MAPING"."PBV-85 SORBITOL INLET LINE" := FALSE;
	    END_IF;
	END_REGION
	
	REGION PBV-86 GLUCOSE INLET LINE
	    IF ("MODE SELECTION DB"."MODE BUFF" = 2 AND "MANUAL BIT"."PBV-86 GLUCOSE INLET LINE")
	        OR ("TRANSFER DB".OUTPUT."PBV-86 GLUCOSE INLET LINE")
	        OR "AUTO SUBOUTPUT DB"."PBV-86 GLUCOSE INLET LINE"
	    THEN
	        "DO MAPING"."PBV-86 GLUCOSE INLET LINE" := TRUE;
	    ELSE
	        "DO MAPING"."PBV-86 GLUCOSE INLET LINE" := FALSE;
	    END_IF;
	END_REGION
	
	REGION PBV-87 BASKET FILTER TO PREMIX VESSEL LINE
	    IF ("MODE SELECTION DB"."MODE BUFF" = 2 AND "MANUAL BIT"."PBV-87 BASKET FILTER TO PREMIX VESSEL LINE")
	        OR ("TRANSFER DB".OUTPUT."PBV-87 BASKET FILTER TO PREMIX VESSEL LINE")
	        OR "AUTO SUBOUTPUT DB"."PBV-87 BASKET FILTER TO PREMIX VESSEL LINE"
	    THEN
	        "DO MAPING"."PBV-87 BASKET FILTER TO PREMIX VESSEL LINE" := TRUE;
	    ELSE
	        "DO MAPING"."PBV-87 BASKET FILTER TO PREMIX VESSEL LINE" := FALSE;
	    END_IF;
	END_REGION
	
	REGION PBV-88 BASKET FILTER TRANSFER LINE
	    IF ("MODE SELECTION DB"."MODE BUFF" = 2 AND "MANUAL BIT"."PBV-88 BASKET FILTER TRANSFER LINE")
	        OR ("TRANSFER DB".OUTPUT."PBV-88 BASKET FILTER TRANSFER LINE")
	        OR "AUTO SUBOUTPUT DB"."PBV-88 BASKET FILTER TRANSFER LINE"
	    THEN
	        "DO MAPING"."PBV-88 BASKET FILTER TRANSFER LINE" := TRUE;
	    ELSE
	        "DO MAPING"."PBV-88 BASKET FILTER TRANSFER LINE" := FALSE;
	    END_IF;
	END_REGION
	
	REGION PBV-89 BASKET FILTER TO MFG INLET TRANSFER LINE
	    IF ("MODE SELECTION DB"."MODE BUFF" = 2 AND "MANUAL BIT"."PBV-89 BASKET FILTER TO MFG INLET TRANSFER LINE")
	        OR ("TRANSFER DB".OUTPUT."PBV-89 BASKET FILTER TO MFG INLET TRANSFER LINE")
	        OR "AUTO SUBOUTPUT DB"."PBV-89 BASKET FILTER TO MFG INLET TRANSFER LINE"
	    THEN
	        "DO MAPING"."PBV-89 BASKET FILTER TO MFG INLET TRANSFER LINE" := TRUE;
	    ELSE
	        "DO MAPING"."PBV-89 BASKET FILTER TO MFG INLET TRANSFER LINE" := FALSE;
	    END_IF;
	END_REGION
	
	REGION PBV-90 PREMIX TO MFG TRANSFER LINE
	    IF ("MODE SELECTION DB"."MODE BUFF" = 2 AND "MANUAL BIT"."PBV-90 PREMIX TO MFG TRANSFER LINE")
	        OR ("TRANSFER DB".OUTPUT."PBV-90 PREMIX TO MFG TRANSFER LINE")
	        OR "AUTO SUBOUTPUT DB"."PBV-90 PREMIX TO MFG TRANSFER LINE"
	    THEN
	        "DO MAPING"."PBV-90 PREMIX TO MFG TRANSFER LINE" := TRUE;
	    ELSE
	        "DO MAPING"."PBV-90 PREMIX TO MFG TRANSFER LINE" := FALSE;
	    END_IF;
	END_REGION
	
	REGION PBV-91 PREMIX TO MFG TRANSFER LINE
	    IF ("MODE SELECTION DB"."MODE BUFF" = 2 AND "MANUAL BIT"."PBV-91 PREMIX TO MFG TRANSFER LINE")
	        OR ("TRANSFER DB".OUTPUT."PBV-91 PREMIX TO MFG TRANSFER LINE")
	        OR "AUTO SUBOUTPUT DB"."PBV-91 PREMIX TO MFG TRANSFER LINE"
	    THEN
	        "DO MAPING"."PBV-91 PREMIX TO MFG TRANSFER LINE" := TRUE;
	    ELSE
	        "DO MAPING"."PBV-91 PREMIX TO MFG TRANSFER LINE" := FALSE;
	    END_IF;
	END_REGION
	
	REGION PBV-92 PREMIX TO STORAGE – 4 TRANSFER LINE
	    IF ("MODE SELECTION DB"."MODE BUFF" = 2 AND "MANUAL BIT"."PBV-92 PREMIX TO STORAGE – 4 TRANSFER LINE")
	        OR ("TRANSFER DB".OUTPUT."PBV-92 PREMIX TO STORAGE – 4 TRANSFER LINE")
	        OR "AUTO SUBOUTPUT DB"."PBV-92 PREMIX TO STORAGE – 4 TRANSFER LINE"
	    THEN
	        "DO MAPING"."PBV-92 PREMIX TO STORAGE – 4 TRANSFER LINE" := TRUE;
	    ELSE
	        "DO MAPING"."PBV-92 PREMIX TO STORAGE – 4 TRANSFER LINE" := FALSE;
	    END_IF;
	END_REGION
	
	REGION PBV-93 TANK OUTLET TO INLINE HOMOGENIZER LINE
	    IF ("MODE SELECTION DB"."MODE BUFF" = 2 AND "MANUAL BIT"."PBV-93 TANK OUTLET TO INLINE HOMOGENIZER LINE")
	        OR ("TRANSFER DB".OUTPUT."PBV-93 TANK OUTLET TO INLINE HOMOGENIZER LINE")
	        OR "AUTO SUBOUTPUT DB"."PBV-93 TANK OUTLET TO INLINE HOMOGENIZER LINE"
	    THEN
	        "DO MAPING"."PBV-93 TANK OUTLET TO INLINE HOMOGENIZER LINE" := TRUE;
	    ELSE
	        "DO MAPING"."PBV-93 TANK OUTLET TO INLINE HOMOGENIZER LINE" := FALSE;
	    END_IF;
	END_REGION
	
	REGION PBV-94 INLINE HOMOGENIZER INLET LINE
	    IF ("MODE SELECTION DB"."MODE BUFF" = 2 AND "MANUAL BIT"."PBV-94 INLINE HOMOGENIZER INLET LINE")
	        OR ("TRANSFER DB".OUTPUT."PBV-94 INLINE HOMOGENIZER INLET LINE")
	        OR "AUTO SUBOUTPUT DB"."PBV-94 INLINE HOMOGENIZER INLET LINE"
	    THEN
	        "DO MAPING"."PBV-94 INLINE HOMOGENIZER INLET LINE" := TRUE;
	    ELSE
	        "DO MAPING"."PBV-94 INLINE HOMOGENIZER INLET LINE" := FALSE;
	    END_IF;
	END_REGION
	
	REGION PBV-95 TANK OUTLET TO FILTER PRESS LINE
	    IF ("MODE SELECTION DB"."MODE BUFF" = 2 AND "MANUAL BIT"."PBV-95 TANK OUTLET TO FILTER PRESS LINE")
	        OR ("TRANSFER DB".OUTPUT."PBV-95 TANK OUTLET TO FILTER PRESS LINE")
	        OR "AUTO SUBOUTPUT DB"."PBV-95 TANK OUTLET TO FILTER PRESS LINE"
	    THEN
	        "DO MAPING"."PBV-95 TANK OUTLET TO FILTER PRESS LINE" := TRUE;
	    ELSE
	        "DO MAPING"."PBV-95 TANK OUTLET TO FILTER PRESS LINE" := FALSE;
	    END_IF;
	END_REGION
	
	REGION PBV-96 INLINE HOMOGENIZER RECIRCULATION LINE
	    IF ("MODE SELECTION DB"."MODE BUFF" = 2 AND "MANUAL BIT"."PBV-96 INLINE HOMOGENIZER RECIRCULATION LINE")
	        OR ("TRANSFER DB".OUTPUT."PBV-96 INLINE HOMOGENIZER RECIRCULATION LINE")
	        OR "AUTO SUBOUTPUT DB"."PBV-96 INLINE HOMOGENIZER RECIRCULATION LINE"
	    THEN
	        "DO MAPING"."PBV-96 INLINE HOMOGENIZER RECIRCULATION LINE" := TRUE;
	    ELSE
	        "DO MAPING"."PBV-96 INLINE HOMOGENIZER RECIRCULATION LINE" := FALSE;
	    END_IF;
	END_REGION
	
	REGION PBV-97 FILTER PRESS OUTLET
	    IF ("MODE SELECTION DB"."MODE BUFF" = 2 AND "MANUAL BIT"."PBV-97 FILTER PRESS OUTLET")
	        OR ("TRANSFER DB".OUTPUT."PBV-97 FILTER PRESS OUTLET")
	        OR "AUTO SUBOUTPUT DB"."PBV-97 FILTER PRESS OUTLET"
	    THEN
	        "DO MAPING"."PBV-97 FILTER PRESS OUTLET" := TRUE;
	    ELSE
	        "DO MAPING"."PBV-97 FILTER PRESS OUTLET" := FALSE;
	    END_IF;
	END_REGION
	
	REGION PBV-98 INLINE HOMOGENIZER TO FILTER PRESS OUTLET LINE
	    IF ("MODE SELECTION DB"."MODE BUFF" = 2 AND "MANUAL BIT"."PBV-98 INLINE HOMOGENIZER TO FILTER PRESS OUTLET LINE")
	        OR ("TRANSFER DB".OUTPUT."PBV-98 INLINE HOMOGENIZER TO FILTER PRESS OUTLET LINE")
	        OR "AUTO SUBOUTPUT DB"."PBV-98 INLINE HOMOGENIZER TO FILTER PRESS OUTLET LINE"
	    THEN
	        "DO MAPING"."PBV-98 INLINE HOMOGENIZER TO FILTER PRESS OUTLET LINE" := TRUE;
	    ELSE
	        "DO MAPING"."PBV-98 INLINE HOMOGENIZER TO FILTER PRESS OUTLET LINE" := FALSE;
	    END_IF;
	END_REGION
	
	REGION PAV-99 INLINE HOMOGENIZER SEAL COOLING
	    IF ("MODE SELECTION DB"."MODE BUFF" = 2 AND "MANUAL BIT"."PAV-99 INLINE HOMOGENIZER SEAL COOLING")
	        OR ("TRANSFER DB".OUTPUT."PAV-99 INLINE HOMOGENIZER SEAL COOLING")
	        OR "AUTO SUBOUTPUT DB"."PAV-99 INLINE HOMOGENIZER SEAL COOLING"
	    THEN
	        "DO MAPING"."PAV-99 INLINE HOMOGENIZER SEAL COOLING" := TRUE;
	    ELSE
	        "DO MAPING"."PAV-99 INLINE HOMOGENIZER SEAL COOLING" := FALSE;
	    END_IF;
	END_REGION
	
	REGION PBV-100 FILTER PRESS INLET
	    IF ("MODE SELECTION DB"."MODE BUFF" = 2 AND "MANUAL BIT"."PBV-100 FILTER PRESS INLET")
	        OR ("TRANSFER DB".OUTPUT."PBV-100 FILTER PRESS INLET")
	        OR "AUTO SUBOUTPUT DB"."PBV-100 FILTER PRESS INLET"
	    THEN
	        "DO MAPING"."PBV-100 FILTER PRESS INLET" := TRUE;
	    ELSE
	        "DO MAPING"."PBV-100 FILTER PRESS INLET" := FALSE;
	    END_IF;
	END_REGION
	
	REGION PBV-101 SUGAR MELTING TO MFG TRANSFER (TOP DISH)
	    IF ("MODE SELECTION DB"."MODE BUFF" = 2 AND "MANUAL BIT"."PBV-101 SUGAR MELTING TO MFG TRANSFER (TOP DISH)")
	        OR ("TRANSFER DB".OUTPUT."PBV-101 SUGAR MELTING TO MFG TRANSFER (TOP DISH)")
	        OR "AUTO SUBOUTPUT DB"."PBV-101 SUGAR MELTING TO MFG TRANSFER (TOP DISH)"
	    THEN
	        "DO MAPING"."PBV-101 SUGAR MELTING TO MFG TRANSFER (TOP DISH)" := TRUE;
	    ELSE
	        "DO MAPING"."PBV-101 SUGAR MELTING TO MFG TRANSFER (TOP DISH)" := FALSE;
	    END_IF;
	END_REGION
	
	REGION PBV-102 PREMIX TO MFG TRANSFER (TOP DISH)
	    IF ("MODE SELECTION DB"."MODE BUFF" = 2 AND "MANUAL BIT"."PBV-102 PREMIX TO MFG TRANSFER (TOP DISH)")
	        OR ("TRANSFER DB".OUTPUT."PBV-102 PREMIX TO MFG TRANSFER (TOP DISH)")
	        OR "AUTO SUBOUTPUT DB"."PBV-102 PREMIX TO MFG TRANSFER (TOP DISH)"
	    THEN
	        "DO MAPING"."PBV-102 PREMIX TO MFG TRANSFER (TOP DISH)" := TRUE;
	    ELSE
	        "DO MAPING"."PBV-102 PREMIX TO MFG TRANSFER (TOP DISH)" := FALSE;
	    END_IF;
	END_REGION
	
	REGION PBV-103 CIP INLET (SPRAY BALL)
	    IF ("MODE SELECTION DB"."MODE BUFF" = 2 AND "MANUAL BIT"."PBV-103 CIP INLET (SPRAY BALL)")
	        OR ("TRANSFER DB".OUTPUT."PBV-103 CIP INLET (SPRAY BALL)")
	        OR "AUTO SUBOUTPUT DB"."PBV-103 CIP INLET (SPRAY BALL)"
	    THEN
	        "DO MAPING"."PBV-103 CIP INLET (SPRAY BALL)" := TRUE;
	    ELSE
	        "DO MAPING"."PBV-103 CIP INLET (SPRAY BALL)" := FALSE;
	    END_IF;
	END_REGION
	
	REGION PBV-104 MFG VESSEL TRANSFER LINE
	    IF ("MODE SELECTION DB"."MODE BUFF" = 2 AND "MANUAL BIT"."PBV-104 MFG VESSEL TRANSFER LINE")
	        OR ("TRANSFER DB".OUTPUT."PBV-104 MFG VESSEL TRANSFER LINE")
	        OR "AUTO SUBOUTPUT DB"."PBV-104 MFG VESSEL TRANSFER LINE"
	    THEN
	        "DO MAPING"."PBV-104 MFG VESSEL TRANSFER LINE" := TRUE;
	    ELSE
	        "DO MAPING"."PBV-104 MFG VESSEL TRANSFER LINE" := FALSE;
	    END_IF;
	END_REGION
	
	REGION PBV-105 INGREDIENT INLET
	    IF ("MODE SELECTION DB"."MODE BUFF" = 2 AND "MANUAL BIT"."PBV-105 INGREDIENT INLET")
	        OR ("TRANSFER DB".OUTPUT."PBV-105 INGREDIENT INLET")
	        OR "AUTO SUBOUTPUT DB"."PBV-105 INGREDIENT INLET"
	    THEN
	        "DO MAPING"."PBV-105 INGREDIENT INLET" := TRUE;
	    ELSE
	        "DO MAPING"."PBV-105 INGREDIENT INLET" := FALSE;
	    END_IF;
	END_REGION
	
	REGION PBV-106 SORBITOL INLET
	    IF ("MODE SELECTION DB"."MODE BUFF" = 2 AND "MANUAL BIT"."PBV-106 SORBITOL INLET")
	        OR ("TRANSFER DB".OUTPUT."PBV-106 SORBITOL INLET")
	        OR "AUTO SUBOUTPUT DB"."PBV-106 SORBITOL INLET"
	    THEN
	        "DO MAPING"."PBV-106 SORBITOL INLET" := TRUE;
	    ELSE
	        "DO MAPING"."PBV-106 SORBITOL INLET" := FALSE;
	    END_IF;
	END_REGION
	
	REGION PBV-107 GLUCOSE INLET
	    IF ("MODE SELECTION DB"."MODE BUFF" = 2 AND "MANUAL BIT"."PBV-107 GLUCOSE INLET")
	        OR ("TRANSFER DB".OUTPUT."PBV-107 GLUCOSE INLET")
	        OR "AUTO SUBOUTPUT DB"."PBV-107 GLUCOSE INLET"
	    THEN
	        "DO MAPING"."PBV-107 GLUCOSE INLET" := TRUE;
	    ELSE
	        "DO MAPING"."PBV-107 GLUCOSE INLET" := FALSE;
	    END_IF;
	END_REGION
	
	REGION PBV-108 INLINE HOMOGENIZER TO FILTER PRESS INLET LINE
	    IF ("MODE SELECTION DB"."MODE BUFF" = 2 AND "MANUAL BIT"."PBV-108 INLINE HOMOGENIZER TO FILTER PRESS INLET LINE")
	        OR ("TRANSFER DB".OUTPUT."PBV-108 INLINE HOMOGENIZER TO FILTER PRESS INLET LINE")
	        OR "AUTO SUBOUTPUT DB"."PBV-108 INLINE HOMOGENIZER TO FILTER PRESS INLET LINE"
	    THEN
	        "DO MAPING"."PBV-108 INLINE HOMOGENIZER TO FILTER PRESS INLET LINE" := TRUE;
	    ELSE
	        "DO MAPING"."PBV-108 INLINE HOMOGENIZER TO FILTER PRESS INLET LINE" := FALSE;
	    END_IF;
	END_REGION
	
	REGION PBV-109 HOMO. RECIRCULATION INLET
	    IF ("MODE SELECTION DB"."MODE BUFF" = 2 AND "MANUAL BIT"."PBV-109 HOMO. RECIRCULATION INLET")
	        OR ("TRANSFER DB".OUTPUT."PBV-109 HOMO. RECIRCULATION INLET")
	        OR "AUTO SUBOUTPUT DB"."PBV-109 HOMO. RECIRCULATION INLET"
	    THEN
	        "DO MAPING"."PBV-109 HOMO. RECIRCULATION INLET" := TRUE;
	    ELSE
	        "DO MAPING"."PBV-109 HOMO. RECIRCULATION INLET" := FALSE;
	    END_IF;
	END_REGION
	
	REGION PBV-110 INLINE HOMOGENIZER TO INLET LINE
	    IF ("MODE SELECTION DB"."MODE BUFF" = 2 AND "MANUAL BIT"."PBV-110 INLINE HOMOGENIZER TO INLET LINE")
	        OR ("TRANSFER DB".OUTPUT."PBV-110 INLINE HOMOGENIZER TO INLET LINE")
	        OR "AUTO SUBOUTPUT DB"."PBV-110 INLINE HOMOGENIZER TO INLET LINE"
	    THEN
	        "DO MAPING"."PBV-110 INLINE HOMOGENIZER TO INLET LINE" := TRUE;
	    ELSE
	        "DO MAPING"."PBV-110 INLINE HOMOGENIZER TO INLET LINE" := FALSE;
	    END_IF;
	END_REGION
	
	REGION PBV-111 FILTER PRESS OUTLER VALVE
	    IF ("MODE SELECTION DB"."MODE BUFF" = 2 AND "MANUAL BIT"."PBV-111 FILTER PRESS OUTLER VALVE")
	        OR ("TRANSFER DB".OUTPUT."PBV-111 FILTER PRESS OUTLER VALVE")
	        OR "AUTO SUBOUTPUT DB"."PBV-111 FILTER PRESS OUTLER VALVE"
	    THEN
	        "DO MAPING"."PBV-111 FILTER PRESS OUTLER VALVE" := TRUE;
	    ELSE
	        "DO MAPING"."PBV-111 FILTER PRESS OUTLER VALVE" := FALSE;
	    END_IF;
	END_REGION
	
	REGION PBV-112 FILTER PRESS TO TRANSFER LINE
	    IF ("MODE SELECTION DB"."MODE BUFF" = 2 AND "MANUAL BIT"."PBV-112 FILTER PRESS TO TRANSFER LINE")
	        OR ("TRANSFER DB".OUTPUT."PBV-112 FILTER PRESS TO TRANSFER LINE")
	        OR "AUTO SUBOUTPUT DB"."PBV-112 FILTER PRESS TO TRANSFER LINE"
	    THEN
	        "DO MAPING"."PBV-112 FILTER PRESS TO TRANSFER LINE" := TRUE;
	    ELSE
	        "DO MAPING"."PBV-112 FILTER PRESS TO TRANSFER LINE" := FALSE;
	    END_IF;
	END_REGION
	
	REGION PAV-113 TANK OUTLET TO CIP DRAIN LINE
	    IF ("MODE SELECTION DB"."MODE BUFF" = 2 AND "MANUAL BIT"."PAV-113 TANK OUTLET TO CIP DRAIN LINE")
	        OR ("TRANSFER DB".OUTPUT."PAV-113 TANK OUTLET TO CIP DRAIN LINE")
	        OR "AUTO SUBOUTPUT DB"."PAV-113 TANK OUTLET TO CIP DRAIN LINE"
	    THEN
	        "DO MAPING"."PAV-113 TANK OUTLET TO CIP DRAIN LINE" := TRUE;
	    ELSE
	        "DO MAPING"."PAV-113 TANK OUTLET TO CIP DRAIN LINE" := FALSE;
	    END_IF;
	END_REGION
	
	REGION PBV-114 TANK OUTLET TO INLINE HOMOGENIZER LINE
	    IF ("MODE SELECTION DB"."MODE BUFF" = 2 AND "MANUAL BIT"."PBV-114 TANK OUTLET TO INLINE HOMOGENIZER LINE")
	        OR ("TRANSFER DB".OUTPUT."PBV-114 TANK OUTLET TO INLINE HOMOGENIZER LINE")
	        OR "AUTO SUBOUTPUT DB"."PBV-114 TANK OUTLET TO INLINE HOMOGENIZER LINE"
	    THEN
	        "DO MAPING"."PBV-114 TANK OUTLET TO INLINE HOMOGENIZER LINE" := TRUE;
	    ELSE
	        "DO MAPING"."PBV-114 TANK OUTLET TO INLINE HOMOGENIZER LINE" := FALSE;
	    END_IF;
	END_REGION
	
	REGION PBV-115 MFG TO STORAGE – 1 TRANSFER LINE
	    IF ("MODE SELECTION DB"."MODE BUFF" = 2 AND "MANUAL BIT"."PBV-115 MFG TO STORAGE – 1 TRANSFER LINE")
	        OR ("TRANSFER DB".OUTPUT."PBV-115 MFG TO STORAGE – 1 TRANSFER LINE")
	        OR "AUTO SUBOUTPUT DB"."PBV-115 MFG TO STORAGE – 1 TRANSFER LINE"
	    THEN
	        "DO MAPING"."PBV-115 MFG TO STORAGE – 1 TRANSFER LINE" := TRUE;
	    ELSE
	        "DO MAPING"."PBV-115 MFG TO STORAGE – 1 TRANSFER LINE" := FALSE;
	    END_IF;
	END_REGION
	
	REGION PBV-116 MFG TO STORAGE – 2 TRANSFER LINE
	    IF ("MODE SELECTION DB"."MODE BUFF" = 2 AND "MANUAL BIT"."PBV-116 MFG TO STORAGE – 2 TRANSFER LINE")
	        OR ("TRANSFER DB".OUTPUT."PBV-116 MFG TO STORAGE – 2 TRANSFER LINE")
	        OR "AUTO SUBOUTPUT DB"."PBV-116 MFG TO STORAGE – 2 TRANSFER LINE"
	    THEN
	        "DO MAPING"."PBV-116 MFG TO STORAGE – 2 TRANSFER LINE" := TRUE;
	    ELSE
	        "DO MAPING"."PBV-116 MFG TO STORAGE – 2 TRANSFER LINE" := FALSE;
	    END_IF;
	END_REGION
	
	REGION PBV-117 MFG TO STORAGE – 3 TRANSFER LINE
	    IF ("MODE SELECTION DB"."MODE BUFF" = 2 AND "MANUAL BIT"."PBV-117 MFG TO STORAGE – 3 TRANSFER LINE")
	        OR ("TRANSFER DB".OUTPUT."PBV-117 MFG TO STORAGE – 3 TRANSFER LINE")
	        OR "AUTO SUBOUTPUT DB"."PBV-117 MFG TO STORAGE – 3 TRANSFER LINE"
	    THEN
	        "DO MAPING"."PBV-117 MFG TO STORAGE – 3 TRANSFER LINE" := TRUE;
	    ELSE
	        "DO MAPING"."PBV-117 MFG TO STORAGE – 3 TRANSFER LINE" := FALSE;
	    END_IF;
	END_REGION
	
	REGION PBV-118 FILTER PRESS INLET
	    IF ("MODE SELECTION DB"."MODE BUFF" = 2 AND "MANUAL BIT"."PBV-118 FILTER PRESS INLET")
	        OR ("TRANSFER DB".OUTPUT."PBV-118 FILTER PRESS INLET")
	        OR "AUTO SUBOUTPUT DB"."PBV-118 FILTER PRESS INLET"
	    THEN
	        "DO MAPING"."PBV-118 FILTER PRESS INLET" := TRUE;
	    ELSE
	        "DO MAPING"."PBV-118 FILTER PRESS INLET" := FALSE;
	    END_IF;
	END_REGION
	
	REGION PBV-119 SEAL COOLING FOR STORAGE VESSEL - 4
	    IF ("MODE SELECTION DB"."MODE BUFF" = 2 AND "MANUAL BIT"."PBV-119 SEAL COOLING FOR STORAGE VESSEL - 4")
	        OR ("TRANSFER DB".OUTPUT."PBV-119 SEAL COOLING FOR STORAGE VESSEL - 4")
	        OR "AUTO SUBOUTPUT DB"."PBV-119 SEAL COOLING FOR STORAGE VESSEL - 4"
	    THEN
	        "DO MAPING"."PBV-119 SEAL COOLING FOR STORAGE VESSEL - 4" := TRUE;
	    ELSE
	        "DO MAPING"."PBV-119 SEAL COOLING FOR STORAGE VESSEL - 4" := FALSE;
	    END_IF;
	END_REGION
	
	REGION PBV-120 SEAL COOLING FOR STORAGE VESSEL - 3
	    IF ("MODE SELECTION DB"."MODE BUFF" = 2 AND "MANUAL BIT"."PBV-120 SEAL COOLING FOR STORAGE VESSEL - 3")
	        OR ("TRANSFER DB".OUTPUT."PBV-120 SEAL COOLING FOR STORAGE VESSEL - 3")
	        OR "AUTO SUBOUTPUT DB"."PBV-120 SEAL COOLING FOR STORAGE VESSEL - 3"
	    THEN
	        "DO MAPING"."PBV-120 SEAL COOLING FOR STORAGE VESSEL - 3" := TRUE;
	    ELSE
	        "DO MAPING"."PBV-120 SEAL COOLING FOR STORAGE VESSEL - 3" := FALSE;
	    END_IF;
	END_REGION
	
	REGION PBV-121 SEAL COOLING FOR STORAGE VESSEL - 2
	    IF ("MODE SELECTION DB"."MODE BUFF" = 2 AND "MANUAL BIT"."PBV-121 SEAL COOLING FOR STORAGE VESSEL - 2")
	        OR ("TRANSFER DB".OUTPUT."PBV-121 SEAL COOLING FOR STORAGE VESSEL - 2")
	        OR "AUTO SUBOUTPUT DB"."PBV-121 SEAL COOLING FOR STORAGE VESSEL - 2"
	    THEN
	        "DO MAPING"."PBV-121 SEAL COOLING FOR STORAGE VESSEL - 2" := TRUE;
	    ELSE
	        "DO MAPING"."PBV-121 SEAL COOLING FOR STORAGE VESSEL - 2" := FALSE;
	    END_IF;
	END_REGION
	
	REGION PBV-122 SEAL COOLING FOR STORAGE VESSEL - 1
	    IF ("MODE SELECTION DB"."MODE BUFF" = 2 AND "MANUAL BIT"."PBV-122 SEAL COOLING FOR STORAGE VESSEL - 1")
	        OR ("TRANSFER DB".OUTPUT."PBV-122 SEAL COOLING FOR STORAGE VESSEL - 1")
	        OR "AUTO SUBOUTPUT DB"."PBV-122 SEAL COOLING FOR STORAGE VESSEL - 1"
	    THEN
	        "DO MAPING"."PBV-122 SEAL COOLING FOR STORAGE VESSEL - 1" := TRUE;
	    ELSE
	        "DO MAPING"."PBV-122 SEAL COOLING FOR STORAGE VESSEL - 1" := FALSE;
	    END_IF;
	END_REGION
	
	REGION PBV-123 VESSEL TOP DISH
	    IF ("MODE SELECTION DB"."MODE BUFF" = 2 AND "MANUAL BIT"."PBV-123 VESSEL TOP DISH")
	        OR ("TRANSFER DB".OUTPUT."PBV-123 VESSEL TOP DISH")
	        OR "AUTO SUBOUTPUT DB"."PBV-123 VESSEL TOP DISH"
	    THEN
	        "DO MAPING"."PBV-123 VESSEL TOP DISH" := TRUE;
	    ELSE
	        "DO MAPING"."PBV-123 VESSEL TOP DISH" := FALSE;
	    END_IF;
	END_REGION
	
	REGION PBV-124 VESSEL INLET LINE
	    IF ("MODE SELECTION DB"."MODE BUFF" = 2 AND "MANUAL BIT"."PBV-124 VESSEL INLET LINE")
	        OR ("TRANSFER DB".OUTPUT."PBV-124 VESSEL INLET LINE")
	        OR "AUTO SUBOUTPUT DB"."PBV-124 VESSEL INLET LINE"
	    THEN
	        "DO MAPING"."PBV-124 VESSEL INLET LINE" := TRUE;
	    ELSE
	        "DO MAPING"."PBV-124 VESSEL INLET LINE" := FALSE;
	    END_IF;
	END_REGION
	
	REGION PBV-149
	    IF ("MODE SELECTION DB"."MODE BUFF" = 2 AND "MANUAL BIT"."PBV-149")
	        OR ("TRANSFER DB".OUTPUT."PBV-149")
	        OR "AUTO SUBOUTPUT DB"."PBV-149"
	    THEN
	        "DO MAPING"."PBV-149" := TRUE;
	    ELSE
	        "DO MAPING"."PBV-149" := FALSE;
	    END_IF;
	END_REGION
	
	REGION PBV-150
	    IF ("MODE SELECTION DB"."MODE BUFF" = 2 AND "MANUAL BIT"."PBV-150")
	        OR ("TRANSFER DB".OUTPUT."PBV-150")
	        OR "AUTO SUBOUTPUT DB"."PBV-150"
	    THEN
	        "DO MAPING"."PBV-150" := TRUE;
	    ELSE
	        "DO MAPING"."PBV-150" := FALSE;
	    END_IF;
	END_REGION
	
	REGION PBV-151
	    IF ("MODE SELECTION DB"."MODE BUFF" = 2 AND "MANUAL BIT"."PBV-151")
	        OR ("TRANSFER DB".OUTPUT."PBV-151")
	        OR "AUTO SUBOUTPUT DB"."PBV-151"
	    THEN
	        "DO MAPING"."PBV-151" := TRUE;
	    ELSE
	        "DO MAPING"."PBV-151" := FALSE;
	    END_IF;
	END_REGION
	
	REGION PBV-152
	    IF ("MODE SELECTION DB"."MODE BUFF" = 2 AND "MANUAL BIT"."PBV-152")
	        OR ("TRANSFER DB".OUTPUT."PBV-152")
	        OR "AUTO SUBOUTPUT DB"."PBV-152"
	    THEN
	        "DO MAPING"."PBV-152" := TRUE;
	    ELSE
	        "DO MAPING"."PBV-152" := FALSE;
	    END_IF;
	END_REGION
	
	REGION PBV-153
	    IF ("MODE SELECTION DB"."MODE BUFF" = 2 AND "MANUAL BIT"."PBV-153")
	        OR ("TRANSFER DB".OUTPUT."PBV-153")
	        OR "AUTO SUBOUTPUT DB"."PBV-153"
	    THEN
	        "DO MAPING"."PBV-153" := TRUE;
	    ELSE
	        "DO MAPING"."PBV-153" := FALSE;
	    END_IF;
	END_REGION
	
	REGION PBV-155
	    IF ("MODE SELECTION DB"."MODE BUFF" = 2 AND "MANUAL BIT"."PBV-155")
	        OR ("TRANSFER DB".OUTPUT."PBV-155")
	        OR "AUTO SUBOUTPUT DB"."PBV-155"
	    THEN
	        "DO MAPING"."PBV-155" := TRUE;
	    ELSE
	        "DO MAPING"."PBV-155" := FALSE;
	    END_IF;
	END_REGION
	
	REGION PBV-155
	    IF ("MODE SELECTION DB"."MODE BUFF" = 2 AND "MANUAL BIT"."PBV-156")
	        OR ("TRANSFER DB".OUTPUT."PBV-156")
	        OR "AUTO SUBOUTPUT DB"."PBV-156"
	    THEN
	        "DO MAPING"."PBV-156" := TRUE;
	    ELSE
	        "DO MAPING"."PBV-156" := FALSE;
	    END_IF;
	END_REGION
	
	
	
	
	
	
	
	
	
	
	
	
	
	
	
	
	
	
	
	
	
	
	
	
	
	
	
	
	
	
	
	
	
	
	
	
	
	
	
	
	
END_FUNCTION

FUNCTION "TRANSFER PROCESS & SET CUTOUT" : Void   // FC12, LAD
{ S7_Optimized_Access := 'TRUE' }
// stored: SetENOAutomatically false
   VAR_TEMP   // added for the SCL form of the ladder/FBD networks
      _w1 : Bool;
      _w2 : Bool;
   END_VAR
BEGIN

REGION Network 1 (SCL): MFG VESSEL STIRRER RUN
   REGION MFG VESSEL STIRRER RUN

       IF ("MANUAL TIME BASE DB"."MFG VESSEL STIRRER RUN".SV = 0) OR
           ("MANUAL BIT"."SYRUP MFG VESSEL BOTTOM STERROR RUN" = 1 AND "TIMER_MIN_DB".DONE)
       THEN
           "MANUAL BIT"."SYRUP MFG VESSEL BOTTOM STERROR RUN" := FALSE;
       ELSE
           "TIMER_MIN_DB"("SET TIME" := "MANUAL TIME BASE DB"."MFG VESSEL STIRRER RUN".SV,
                          RESET := "TIMER_MIN_DB".RESET,
                          INPUT := "MANUAL BIT"."SYRUP MFG VESSEL BOTTOM STERROR RUN",
                          "PRESENT VALUE OF TIME" => "MANUAL TIME BASE DB"."MFG VESSEL STIRRER RUN".PV);
       END_IF;
       IF "MODE SELECTION DB"."MODE BUFF" <> 2 OR
           "MANUAL TIME BASE DB"."MFG VESSEL STIRRER RUN"."RESET TIME" = TRUE THEN
           "TIMER_MIN_DB".RESET := TRUE;
       ELSE
           "TIMER_MIN_DB".RESET := FALSE;
       END_IF;
   END_REGION
END_REGION

REGION Network 2 (SCL): PREMIXING VESSEL STIRRER RUN
   REGION PREMIXING  VESSEL STIRRER RUN

       IF ("MANUAL TIME BASE DB"."PREMIXING  VESSEL STIRRER RUN".SV = 0) OR
           ("MANUAL BIT"."PREMIXING VESSEL BOTTOM STERROR RUN" = 1 AND "TIMER_MIN_DB_1".DONE)
       THEN
           "MANUAL BIT"."PREMIXING VESSEL BOTTOM STERROR RUN" := FALSE;
       ELSE
           "TIMER_MIN_DB_1"("SET TIME" := "MANUAL TIME BASE DB"."PREMIXING  VESSEL STIRRER RUN".SV,
                            RESET := "TIMER_MIN_DB_1".RESET,
                            INPUT := "MANUAL BIT"."PREMIXING VESSEL BOTTOM STERROR RUN",
                            "PRESENT VALUE OF TIME" => "MANUAL TIME BASE DB"."PREMIXING  VESSEL STIRRER RUN".PV);
       END_IF;
       IF "MODE SELECTION DB"."MODE BUFF" <> 2 OR
           "MANUAL TIME BASE DB"."PREMIXING  VESSEL STIRRER RUN"."RESET TIME" = TRUE THEN
           "TIMER_MIN_DB_1".RESET := TRUE;
       ELSE
           "TIMER_MIN_DB_1".RESET := FALSE;
       END_IF;
   END_REGION
END_REGION

REGION Network 3 (SCL): SUGAR VESSEL STIRRER RUN
   REGION SUGAR VESSEL STIRRER RUN

       IF ("MANUAL TIME BASE DB"."SUGAR VESSEL STIRRER RUN".SV = 0) OR
           ("MANUAL BIT"."SUGAR VESSEL BOTTOM STERROR RUN" = 1 AND "TIMER_MIN_DB_2".DONE)
       THEN
           "MANUAL BIT"."SUGAR VESSEL BOTTOM STERROR RUN" := FALSE;
       ELSE
           "TIMER_MIN_DB_2"("SET TIME" := "MANUAL TIME BASE DB"."SUGAR VESSEL STIRRER RUN".SV,
                            RESET := "TIMER_MIN_DB_2".RESET,
                            INPUT := "MANUAL BIT"."SUGAR VESSEL BOTTOM STERROR RUN",
                            "PRESENT VALUE OF TIME" => "MANUAL TIME BASE DB"."SUGAR VESSEL STIRRER RUN".PV);
       END_IF;
       IF "MODE SELECTION DB"."MODE BUFF" <> 2 OR
           "MANUAL TIME BASE DB"."SUGAR VESSEL STIRRER RUN"."RESET TIME" = TRUE THEN
           "TIMER_MIN_DB_2".RESET := TRUE;
       ELSE
           "TIMER_MIN_DB_2".RESET := FALSE;
       END_IF;
   END_REGION
END_REGION

REGION Network 5: SYRUP MFG_TEMP_CUTOUT
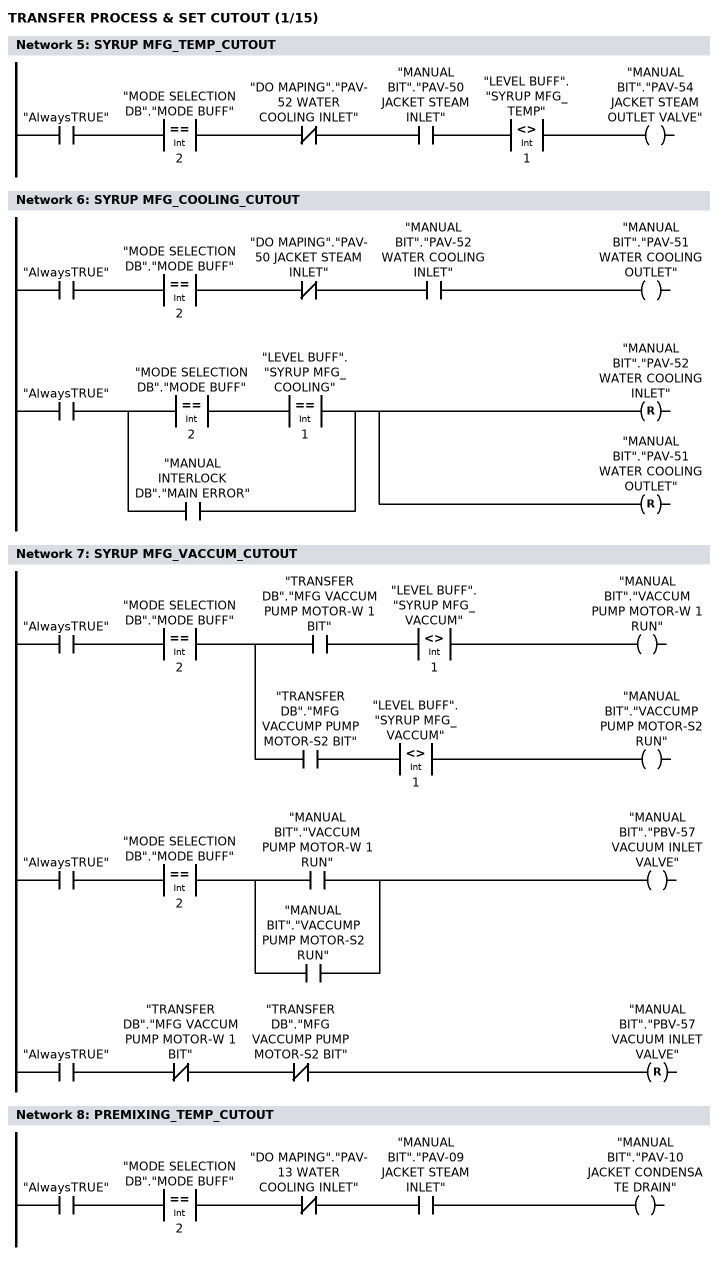
   RUNG wire#powerrail
      Contact( "AlwaysTRUE" )
      { S7_Templates := "SrcType := Int" } EQ_Contact(in1 := "MODE SELECTION DB"."MODE BUFF", in2 := 2)
      I_Contact( "DO MAPING"."PAV-52 WATER COOLING INLET" )
      Contact( "MANUAL BIT"."PAV-50 JACKET STEAM INLET" )
      { S7_Templates := "SrcType := Int" } NE_Contact(in1 := "LEVEL BUFF"."SYRUP MFG_TEMP", in2 := 1)
      Coil( "MANUAL BIT"."PAV-54 JACKET STEAM OUTLET VALVE" )
   END_RUNG
   // the same network as SCL:
   "MANUAL BIT"."PAV-54 JACKET STEAM OUTLET VALVE" := "AlwaysTRUE" AND ("MODE SELECTION DB"."MODE BUFF" = 2) AND NOT "DO MAPING"."PAV-52 WATER COOLING INLET" AND "MANUAL BIT"."PAV-50 JACKET STEAM INLET" AND ("LEVEL BUFF"."SYRUP MFG_TEMP" <> 1);
END_REGION

REGION Network 6: SYRUP MFG_COOLING_CUTOUT
   RUNG wire#powerrail
      Contact( "AlwaysTRUE" )
      { S7_Templates := "SrcType := Int" } EQ_Contact(in1 := "MODE SELECTION DB"."MODE BUFF", in2 := 2)
      I_Contact( "DO MAPING"."PAV-50 JACKET STEAM INLET" )
      Contact( "MANUAL BIT"."PAV-52 WATER COOLING INLET" )
      Coil( "MANUAL BIT"."PAV-51 WATER COOLING OUTLET" )
   END_RUNG
   RUNG wire#powerrail
      Contact( "AlwaysTRUE" )
      wire#w1
      { S7_Templates := "SrcType := Int" } EQ_Contact(in1 := "MODE SELECTION DB"."MODE BUFF", in2 := 2)
      { S7_Templates := "SrcType := Int" } EQ_Contact(in1 := "LEVEL BUFF"."SYRUP MFG_COOLING", in2 := 1)
      wire#w2
      R_Coil( "MANUAL BIT"."PAV-52 WATER COOLING INLET" )
   END_RUNG
   RUNG wire#w1
      Contact( "MANUAL INTERLOCK DB"."MAIN ERROR" )
   END_RUNG wire#w2
   RUNG wire#w2
      R_Coil( "MANUAL BIT"."PAV-51 WATER COOLING OUTLET" )
   END_RUNG
   // the same network as SCL:
   "MANUAL BIT"."PAV-51 WATER COOLING OUTLET" := "AlwaysTRUE" AND ("MODE SELECTION DB"."MODE BUFF" = 2) AND NOT "DO MAPING"."PAV-50 JACKET STEAM INLET" AND "MANUAL BIT"."PAV-52 WATER COOLING INLET";
   IF "AlwaysTRUE" AND ((("MODE SELECTION DB"."MODE BUFF" = 2) AND ("LEVEL BUFF"."SYRUP MFG_COOLING" = 1)) OR "MANUAL INTERLOCK DB"."MAIN ERROR") THEN
       "MANUAL BIT"."PAV-52 WATER COOLING INLET" := FALSE;
       "MANUAL BIT"."PAV-51 WATER COOLING OUTLET" := FALSE;
   END_IF;
END_REGION

REGION Network 7: SYRUP MFG_VACCUM_CUTOUT
   RUNG wire#powerrail
      Contact( "AlwaysTRUE" )
      { S7_Templates := "SrcType := Int" } EQ_Contact(in1 := "MODE SELECTION DB"."MODE BUFF", in2 := 2)
      wire#w1
      Contact( "TRANSFER DB"."MFG VACCUM PUMP MOTOR-W 1 BIT" )
      { S7_Templates := "SrcType := Int" } NE_Contact(in1 := "LEVEL BUFF"."SYRUP MFG_VACCUM", in2 := 1)
      Coil( "MANUAL BIT"."VACCUM PUMP MOTOR-W 1 RUN" )
   END_RUNG
   RUNG wire#w1
      Contact( "TRANSFER DB"."MFG VACCUMP PUMP MOTOR-S2 BIT" )
      { S7_Templates := "SrcType := Int" } NE_Contact(in1 := "LEVEL BUFF"."SYRUP MFG_VACCUM", in2 := 1)
      Coil( "MANUAL BIT"."VACCUMP PUMP MOTOR-S2 RUN" )
   END_RUNG
   RUNG wire#powerrail
      Contact( "AlwaysTRUE" )
      { S7_Templates := "SrcType := Int" } EQ_Contact(in1 := "MODE SELECTION DB"."MODE BUFF", in2 := 2)
      wire#w2
      Contact( "MANUAL BIT"."VACCUM PUMP MOTOR-W 1 RUN" )
      wire#w3
      Coil( "MANUAL BIT"."PBV-57 VACUUM INLET VALVE" )
   END_RUNG
   RUNG wire#w2
      Contact( "MANUAL BIT"."VACCUMP PUMP MOTOR-S2 RUN" )
   END_RUNG wire#w3
   RUNG wire#powerrail
      Contact( "AlwaysTRUE" )
      I_Contact( "TRANSFER DB"."MFG VACCUM PUMP MOTOR-W 1 BIT" )
      I_Contact( "TRANSFER DB"."MFG VACCUMP PUMP MOTOR-S2 BIT" )
      R_Coil( "MANUAL BIT"."PBV-57 VACUUM INLET VALVE" )
   END_RUNG
   // the same network as SCL:
   #_w1 := "AlwaysTRUE" AND ("MODE SELECTION DB"."MODE BUFF" = 2);
   "MANUAL BIT"."VACCUM PUMP MOTOR-W 1 RUN" := #_w1 AND "TRANSFER DB"."MFG VACCUM PUMP MOTOR-W 1 BIT" AND ("LEVEL BUFF"."SYRUP MFG_VACCUM" <> 1);
   "MANUAL BIT"."VACCUMP PUMP MOTOR-S2 RUN" := #_w1 AND "TRANSFER DB"."MFG VACCUMP PUMP MOTOR-S2 BIT" AND ("LEVEL BUFF"."SYRUP MFG_VACCUM" <> 1);
   "MANUAL BIT"."PBV-57 VACUUM INLET VALVE" := "AlwaysTRUE" AND ("MODE SELECTION DB"."MODE BUFF" = 2) AND ("MANUAL BIT"."VACCUM PUMP MOTOR-W 1 RUN" OR "MANUAL BIT"."VACCUMP PUMP MOTOR-S2 RUN");
   IF "AlwaysTRUE" AND NOT "TRANSFER DB"."MFG VACCUM PUMP MOTOR-W 1 BIT" AND NOT "TRANSFER DB"."MFG VACCUMP PUMP MOTOR-S2 BIT" THEN
       "MANUAL BIT"."PBV-57 VACUUM INLET VALVE" := FALSE;
   END_IF;
END_REGION

